   DATA[1132,29] := 12.07383;
   DATA[1132,30] := 1.724686;
   DATA[1132,31] := 1.274753;
   DATA[1132,32] := 0.7352687;
   DATA[1132,33] := 0.3084265;
   DATA[1132,34] := 2.0;
   DATA[1132,35] := 250.1442;
   DATA[1132,36] := 1.537821;
   DATA[1132,37] := 188.958;
   DATA[1132,38] := 0.000128152;
   DATA[1132,39] := 1.0;
   DATA[1133,0] := 2.551965;
   DATA[1133,1] := 721.1517;
   DATA[1133,2] := 2.0;
   DATA[1133,3] := 1.0;
   DATA[1133,4] := 262.5288;
   DATA[1133,5] := 8.463728;
   DATA[1133,6] := 316.7649;
   DATA[1133,8] := 1.0;
   DATA[1133,9] := 1.0;
   DATA[1133,10] := 1.0;
   DATA[1133,11] := 2.010372;
   DATA[1133,12] := 0.000256221;
   DATA[1133,13] := 1010.718;
   DATA[1133,14] := 1.0;
   DATA[1133,15] := 1.0;
   DATA[1133,16] := 1.0;
   DATA[1133,17] := 1.0;
   DATA[1133,18] := 1.0;
   DATA[1133,19] := 1.0;
   DATA[1133,20] := 148.808;
   DATA[1133,21] := 154.3963;
   DATA[1133,22] := 1.709672;
   DATA[1133,23] := 865.2397;
   DATA[1133,24] := 2.0;
   DATA[1133,25] := 2.0;
   DATA[1133,26] := 7.87798;
   DATA[1133,27] := 143.6042;
   DATA[1133,28] := 263.0095;
   DATA[1133,29] := 12.07383;
   DATA[1133,30] := 1.725455;
   DATA[1133,31] := 1.282567;
   DATA[1133,32] := 0.7352687;
   DATA[1133,33] := 0.3084265;
   DATA[1133,34] := 2.0;
   DATA[1133,35] := 250.1442;
   DATA[1133,36] := 1.69801;
   DATA[1133,37] := 189.1022;
   DATA[1133,38] := 0.000128152;
   DATA[1133,39] := 1.0;
   DATA[1134,0] := 2.548762;
   DATA[1134,1] := 722.604;
   DATA[1134,2] := 2.0;
   DATA[1134,3] := 1.0;
   DATA[1134,4] := 262.5288;
   DATA[1134,5] := 8.463728;
   DATA[1134,6] := 316.7649;
   DATA[1134,8] := 1.0;
   DATA[1134,9] := 1.0;
   DATA[1134,10] := 1.0;
   DATA[1134,11] := 2.010372;
   DATA[1134,12] := 0.000256221;
   DATA[1134,13] := 1010.959;
   DATA[1134,14] := 1.0;
   DATA[1134,15] := 1.0;
   DATA[1134,16] := 1.0;
   DATA[1134,17] := 1.0;
   DATA[1134,18] := 1.0;
   DATA[1134,19] := 1.0;
   DATA[1134,20] := 148.808;
   DATA[1134,21] := 154.3963;
   DATA[1134,22] := 1.709672;
   DATA[1134,23] := 865.1628;
   DATA[1134,24] := 2.0;
   DATA[1134,25] := 2.0;
   DATA[1134,26] := 7.87798;
   DATA[1134,27] := 143.6042;
   DATA[1134,28] := 263.0095;
   DATA[1134,29] := 12.07383;
   DATA[1134,30] := 1.725455;
   DATA[1134,31] := 1.282567;
   DATA[1134,32] := 0.7352687;
   DATA[1134,33] := 0.3084265;
   DATA[1134,34] := 2.0;
   DATA[1134,35] := 250.3044;
   DATA[1134,36] := 1.69801;
   DATA[1134,37] := 189.1662;
   DATA[1134,38] := 0.000128152;
   DATA[1134,39] := 1.0;
   DATA[1135,0] := 2.548762;
   DATA[1135,1] := 722.761;
   DATA[1135,2] := 2.0;
   DATA[1135,3] := 1.0;
   DATA[1135,4] := 262.5288;
   DATA[1135,5] := 8.463728;
   DATA[1135,6] := 316.7649;
   DATA[1135,8] := 1.0;
   DATA[1135,9] := 1.0;
   DATA[1135,10] := 1.0;
   DATA[1135,11] := 2.010372;
   DATA[1135,12] := 0.000256221;
   DATA[1135,13] := 1010.839;
   DATA[1135,14] := 1.0;
   DATA[1135,15] := 1.0;
   DATA[1135,16] := 1.0;
   DATA[1135,17] := 1.0;
   DATA[1135,18] := 1.0;
   DATA[1135,19] := 1.0;
   DATA[1135,20] := 148.808;
   DATA[1135,21] := 154.3963;
   DATA[1135,22] := 1.709672;
   DATA[1135,23] := 864.7398;
   DATA[1135,24] := 2.0;
   DATA[1135,25] := 2.0;
   DATA[1135,26] := 7.87798;
   DATA[1135,27] := 143.6042;
   DATA[1135,28] := 263.0095;
   DATA[1135,29] := 12.07383;
   DATA[1135,30] := 1.725455;
   DATA[1135,31] := 1.289484;
   DATA[1135,32] := 0.7352687;
   DATA[1135,33] := 0.3084265;
   DATA[1135,34] := 2.0;
   DATA[1135,35] := 250.3044;
   DATA[1135,36] := 1.69801;
   DATA[1135,37] := 189.1662;
   DATA[1135,38] := 0.000128152;
   DATA[1135,39] := 1.0;
   DATA[1136,0] := 2.548762;
   DATA[1136,1] := 723.4283;
   DATA[1136,2] := 2.0;
   DATA[1136,3] := 1.0;
   DATA[1136,4] := 262.5288;
   DATA[1136,5] := 8.463728;
   DATA[1136,6] := 316.97;
   DATA[1136,8] := 1.0;
   DATA[1136,9] := 1.0;
   DATA[1136,10] := 1.0;
   DATA[1136,11] := 2.010372;
   DATA[1136,12] := 0.000256221;
   DATA[1136,13] := 1011.039;
   DATA[1136,14] := 1.0;
   DATA[1136,15] := 1.0;
   DATA[1136,16] := 1.0;
   DATA[1136,17] := 1.0;
   DATA[1136,18] := 1.0;
   DATA[1136,19] := 1.0;
   DATA[1136,20] := 148.808;
   DATA[1136,21] := 154.3963;
   DATA[1136,22] := 1.709672;
   DATA[1136,23] := 864.586;
   DATA[1136,24] := 2.0;
   DATA[1136,25] := 2.0;
   DATA[1136,26] := 7.87798;
   DATA[1136,27] := 143.6042;
   DATA[1136,28] := 263.0095;
   DATA[1136,29] := 12.07383;
   DATA[1136,30] := 1.725455;
   DATA[1136,31] := 1.29243;
   DATA[1136,32] := 0.7352687;
   DATA[1136,33] := 0.3084265;
   DATA[1136,34] := 2.0;
   DATA[1136,35] := 250.3204;
   DATA[1136,36] := 1.69801;
   DATA[1136,37] := 189.1662;
   DATA[1136,38] := 0.000128152;
   DATA[1136,39] := 1.0;
   DATA[1137,0] := 2.548762;
   DATA[1137,1] := 723.8994;
   DATA[1137,2] := 2.0;
   DATA[1137,3] := 1.0;
   DATA[1137,4] := 262.5288;
   DATA[1137,5] := 8.463728;
   DATA[1137,6] := 316.97;
   DATA[1137,8] := 1.0;
   DATA[1137,9] := 1.0;
   DATA[1137,10] := 1.0;
   DATA[1137,11] := 2.010372;
   DATA[1137,12] := 0.000256221;
   DATA[1137,13] := 1010.959;
   DATA[1137,14] := 1.0;
   DATA[1137,15] := 1.0;
   DATA[1137,16] := 1.0;
   DATA[1137,17] := 1.0;
   DATA[1137,18] := 1.0;
   DATA[1137,19] := 1.0;
   DATA[1137,20] := 148.808;
   DATA[1137,21] := 154.3963;
   DATA[1137,22] := 1.712748;
   DATA[1137,23] := 864.0861;
   DATA[1137,24] := 2.0;
   DATA[1137,25] := 2.0;
   DATA[1137,26] := 7.87798;
   DATA[1137,27] := 143.6042;
   DATA[1137,28] := 263.0095;
   DATA[1137,29] := 12.07383;
   DATA[1137,30] := 1.725455;
   DATA[1137,31] := 1.29243;
   DATA[1137,32] := 0.7352687;
   DATA[1137,33] := 0.3084265;
   DATA[1137,34] := 2.0;
   DATA[1137,35] := 250.3204;
   DATA[1137,36] := 1.69801;
   DATA[1137,37] := 189.1662;
   DATA[1137,38] := 0.000128152;
   DATA[1137,39] := 1.0;
   DATA[1138,0] := 2.550364;
   DATA[1138,1] := 723.7424;
   DATA[1138,2] := 2.0;
   DATA[1138,3] := 1.0;
   DATA[1138,4] := 262.5288;
   DATA[1138,5] := 8.463728;
   DATA[1138,6] := 316.97;
   DATA[1138,8] := 1.0;
   DATA[1138,9] := 1.0;
   DATA[1138,10] := 1.0;
   DATA[1138,11] := 2.010372;
   DATA[1138,12] := 0.000256221;
   DATA[1138,13] := 1010.959;
   DATA[1138,14] := 1.0;
   DATA[1138,15] := 1.0;
   DATA[1138,16] := 1.0;
   DATA[1138,17] := 1.0;
   DATA[1138,18] := 1.0;
   DATA[1138,19] := 1.0;
   DATA[1138,20] := 148.808;
   DATA[1138,21] := 154.3963;
   DATA[1138,22] := 1.713389;
   DATA[1138,23] := 863.817;
   DATA[1138,24] := 2.0;
   DATA[1138,25] := 2.0;
   DATA[1138,26] := 7.87798;
   DATA[1138,27] := 143.6042;
   DATA[1138,28] := 263.0095;
   DATA[1138,29] := 12.07383;
   DATA[1138,30] := 1.725455;
   DATA[1138,31] := 1.285641;
   DATA[1138,32] := 0.7352687;
   DATA[1138,33] := 0.3084265;
   DATA[1138,34] := 2.0;
   DATA[1138,35] := 250.3204;
   DATA[1138,36] := 1.69801;
   DATA[1138,37] := 189.1662;
   DATA[1138,38] := 0.000128152;
   DATA[1138,39] := 1.0;
   DATA[1139,0] := 2.556449;
   DATA[1139,1] := 723.9386;
   DATA[1139,2] := 2.0;
   DATA[1139,3] := 1.0;
   DATA[1139,4] := 262.5288;
   DATA[1139,5] := 8.463728;
   DATA[1139,6] := 316.97;
   DATA[1139,8] := 1.0;
   DATA[1139,9] := 1.0;
   DATA[1139,10] := 1.0;
   DATA[1139,11] := 2.010372;
   DATA[1139,12] := 0.000256221;
   DATA[1139,13] := 1010.638;
   DATA[1139,14] := 1.0;
   DATA[1139,15] := 1.0;
   DATA[1139,16] := 1.0;
   DATA[1139,17] := 1.0;
   DATA[1139,18] := 1.0;
   DATA[1139,19] := 1.0;
   DATA[1139,20] := 148.808;
   DATA[1139,21] := 154.3963;
   DATA[1139,22] := 1.713389;
   DATA[1139,23] := 863.1248;
   DATA[1139,24] := 2.0;
   DATA[1139,25] := 2.0;
   DATA[1139,26] := 7.87798;
   DATA[1139,27] := 143.6042;
   DATA[1139,28] := 263.0095;
   DATA[1139,29] := 12.07383;
   DATA[1139,30] := 1.725455;
   DATA[1139,31] := 1.282311;
   DATA[1139,32] := 0.7352687;
   DATA[1139,33] := 0.3084265;
   DATA[1139,34] := 2.0;
   DATA[1139,35] := 250.2724;
   DATA[1139,36] := 1.69801;
   DATA[1139,37] := 189.0541;
   DATA[1139,38] := 0.000128152;
   DATA[1139,39] := 1.0;
   DATA[1140,0] := 2.560292;
   DATA[1140,1] := 724.9199;
   DATA[1140,2] := 2.0;
   DATA[1140,3] := 1.0;
   DATA[1140,4] := 262.5288;
   DATA[1140,5] := 8.463728;
   DATA[1140,6] := 316.97;
   DATA[1140,8] := 1.0;
   DATA[1140,9] := 1.0;
   DATA[1140,10] := 1.0;
   DATA[1140,11] := 2.010372;
   DATA[1140,12] := 0.000256221;
   DATA[1140,13] := 1011.039;
   DATA[1140,14] := 1.0;
   DATA[1140,15] := 1.0;
   DATA[1140,16] := 1.0;
   DATA[1140,17] := 1.0;
   DATA[1140,18] := 1.0;
   DATA[1140,19] := 1.0;
   DATA[1140,20] := 148.808;
   DATA[1140,21] := 154.3963;
   DATA[1140,22] := 1.713389;
   DATA[1140,23] := 862.8172;
   DATA[1140,24] := 2.0;
   DATA[1140,25] := 2.0;
   DATA[1140,26] := 7.87798;
   DATA[1140,27] := 143.6042;
   DATA[1140,28] := 263.0095;
   DATA[1140,29] := 12.07383;
   DATA[1140,30] := 1.725455;
   DATA[1140,31] := 1.264891;
   DATA[1140,32] := 0.7352687;
   DATA[1140,33] := 0.3084265;
   DATA[1140,34] := 2.0;
   DATA[1140,35] := 250.1762;
   DATA[1140,36] := 1.69801;
   DATA[1140,37] := 189.0541;
   DATA[1140,38] := 0.000128152;
   DATA[1140,39] := 1.0;
   DATA[1141,0] := 2.560292;
   DATA[1141,1] := 725.1555;
   DATA[1141,2] := 2.0;
   DATA[1141,3] := 1.0;
   DATA[1141,4] := 262.5288;
   DATA[1141,5] := 8.463728;
   DATA[1141,6] := 316.97;
   DATA[1141,8] := 1.0;
   DATA[1141,9] := 1.0;
   DATA[1141,10] := 1.0;
   DATA[1141,11] := 2.010372;
   DATA[1141,12] := 0.000256221;
   DATA[1141,13] := 1010.678;
   DATA[1141,14] := 1.0;
   DATA[1141,15] := 1.0;
   DATA[1141,16] := 1.0;
   DATA[1141,17] := 1.0;
   DATA[1141,18] := 1.0;
   DATA[1141,19] := 1.0;
   DATA[1141,20] := 148.808;
   DATA[1141,21] := 154.3963;
   DATA[1141,22] := 1.713389;
   DATA[1141,23] := 862.548;
   DATA[1141,24] := 2.0;
   DATA[1141,25] := 2.0;
   DATA[1141,26] := 7.87798;
   DATA[1141,27] := 143.6042;
   DATA[1141,28] := 263.0095;
   DATA[1141,29] := 12.07383;
   DATA[1141,30] := 1.725455;
   DATA[1141,31] := 1.264634;
   DATA[1141,32] := 0.7352687;
   DATA[1141,33] := 0.3084265;
   DATA[1141,34] := 2.0;
   DATA[1141,35] := 250.1762;
   DATA[1141,36] := 1.69801;
   DATA[1141,37] := 189.0541;
   DATA[1141,38] := 0.000128152;
   DATA[1141,39] := 1.0;
   DATA[1142,0] := 2.560292;
   DATA[1142,1] := 725.7835;
   DATA[1142,2] := 2.0;
   DATA[1142,3] := 1.0;
   DATA[1142,4] := 262.5288;
   DATA[1142,5] := 8.463728;
   DATA[1142,6] := 316.97;
   DATA[1142,8] := 1.0;
   DATA[1142,9] := 1.0;
   DATA[1142,10] := 1.0;
   DATA[1142,11] := 2.010372;
   DATA[1142,12] := 0.000256221;
   DATA[1142,13] := 1011.119;
   DATA[1142,14] := 1.0;
   DATA[1142,15] := 1.0;
   DATA[1142,16] := 1.0;
   DATA[1142,17] := 1.0;
   DATA[1142,18] := 1.0;
   DATA[1142,19] := 1.0;
   DATA[1142,20] := 148.808;
   DATA[1142,21] := 154.3963;
   DATA[1142,22] := 1.714029;
   DATA[1142,23] := 862.0867;
   DATA[1142,24] := 2.0;
   DATA[1142,25] := 2.0;
   DATA[1142,26] := 7.87798;
   DATA[1142,27] := 143.6042;
   DATA[1142,28] := 263.0095;
   DATA[1142,29] := 12.07383;
   DATA[1142,30] := 1.725455;
   DATA[1142,31] := 1.272064;
   DATA[1142,32] := 0.7352687;
   DATA[1142,33] := 0.3084265;
   DATA[1142,34] := 2.0;
   DATA[1142,35] := 250.3204;
   DATA[1142,36] := 1.69801;
   DATA[1142,37] := 189.0541;
   DATA[1142,38] := 0.000128152;
   DATA[1142,39] := 1.0;
   DATA[1143,0] := 2.560292;
   DATA[1143,1] := 726.4901;
   DATA[1143,2] := 2.0;
   DATA[1143,3] := 1.0;
   DATA[1143,4] := 262.5288;
   DATA[1143,5] := 8.463728;
   DATA[1143,6] := 316.9187;
   DATA[1143,8] := 1.0;
   DATA[1143,9] := 1.0;
   DATA[1143,10] := 1.0;
   DATA[1143,11] := 2.010372;
   DATA[1143,12] := 0.000256221;
   DATA[1143,13] := 1011.159;
   DATA[1143,14] := 1.0;
   DATA[1143,15] := 1.0;
   DATA[1143,16] := 1.0;
   DATA[1143,17] := 1.0;
   DATA[1143,18] := 1.0;
   DATA[1143,19] := 1.0;
   DATA[1143,20] := 148.808;
   DATA[1143,21] := 154.3963;
   DATA[1143,22] := 1.714798;
   DATA[1143,23] := 862.0867;
   DATA[1143,24] := 2.0;
   DATA[1143,25] := 2.0;
   DATA[1143,26] := 7.87798;
   DATA[1143,27] := 143.6042;
   DATA[1143,28] := 263.0095;
   DATA[1143,29] := 12.07383;
   DATA[1143,30] := 1.725455;
   DATA[1143,31] := 1.272064;
   DATA[1143,32] := 0.7357808;
   DATA[1143,33] := 0.3084265;
   DATA[1143,34] := 2.0;
   DATA[1143,35] := 250.3365;
   DATA[1143,36] := 1.69801;
   DATA[1143,37] := 189.1823;
   DATA[1143,38] := 0.000128152;
   DATA[1143,39] := 1.0;
   DATA[1144,0] := 2.551324;
   DATA[1144,1] := 726.9218;
   DATA[1144,2] := 2.0;
   DATA[1144,3] := 1.0;
   DATA[1144,4] := 262.5288;
   DATA[1144,5] := 8.463728;
   DATA[1144,6] := 316.7649;
   DATA[1144,8] := 1.0;
   DATA[1144,9] := 1.0;
   DATA[1144,10] := 1.0;
   DATA[1144,11] := 2.010372;
   DATA[1144,12] := 0.000256221;
   DATA[1144,13] := 1011.279;
   DATA[1144,14] := 1.0;
   DATA[1144,15] := 1.0;
   DATA[1144,16] := 1.0;
   DATA[1144,17] := 1.0;
   DATA[1144,18] := 1.0;
   DATA[1144,19] := 1.0;
   DATA[1144,20] := 148.808;
   DATA[1144,21] := 154.3963;
   DATA[1144,22] := 1.714029;
   DATA[1144,23] := 861.6252;
   DATA[1144,24] := 2.0;
   DATA[1144,25] := 2.0;
   DATA[1144,26] := 7.87798;
   DATA[1144,27] := 143.6042;
   DATA[1144,28] := 263.0095;
   DATA[1144,29] := 12.07383;
   DATA[1144,30] := 1.725455;
   DATA[1144,31] := 1.288075;
   DATA[1144,32] := 0.7379573;
   DATA[1144,33] := 0.3084265;
   DATA[1144,34] := 2.0;
   DATA[1144,35] := 250.3365;
   DATA[1144,36] := 1.69801;
   DATA[1144,37] := 189.3265;
   DATA[1144,38] := 0.000128152;
   DATA[1144,39] := 1.0;
   DATA[1145,0] := 2.544919;
   DATA[1145,1] := 727.3143;
   DATA[1145,2] := 2.0;
   DATA[1145,3] := 1.0;
   DATA[1145,4] := 262.5288;
   DATA[1145,5] := 8.463728;
   DATA[1145,6] := 316.7649;
   DATA[1145,8] := 1.0;
   DATA[1145,9] := 1.0;
   DATA[1145,10] := 1.0;
   DATA[1145,11] := 2.010372;
   DATA[1145,12] := 0.000256221;
   DATA[1145,13] := 1011.279;
   DATA[1145,14] := 1.0;
   DATA[1145,15] := 1.0;
   DATA[1145,16] := 1.0;
   DATA[1145,17] := 1.0;
   DATA[1145,18] := 1.0;
   DATA[1145,19] := 1.0;
   DATA[1145,20] := 148.808;
   DATA[1145,21] := 154.3963;
   DATA[1145,22] := 1.713261;
   DATA[1145,23] := 861.3945;
   DATA[1145,24] := 2.0;
   DATA[1145,25] := 2.0;
   DATA[1145,26] := 7.87798;
   DATA[1145,27] := 143.6042;
   DATA[1145,28] := 263.0095;
   DATA[1145,29] := 12.07383;
   DATA[1145,30] := 1.725711;
   DATA[1145,31] := 1.28641;
   DATA[1145,32] := 0.7379573;
   DATA[1145,33] := 0.3084265;
   DATA[1145,34] := 2.0;
   DATA[1145,35] := 250.3365;
   DATA[1145,36] := 1.69801;
   DATA[1145,37] := 189.3265;
   DATA[1145,38] := 0.000128152;
   DATA[1145,39] := 1.0;
   DATA[1146,0] := 2.539154;
   DATA[1146,1] := 727.9424;
   DATA[1146,2] := 2.0;
   DATA[1146,3] := 1.0;
   DATA[1146,4] := 262.5288;
   DATA[1146,5] := 8.463728;
   DATA[1146,6] := 316.7649;
   DATA[1146,8] := 1.0;
   DATA[1146,9] := 1.0;
   DATA[1146,10] := 1.0;
   DATA[1146,11] := 2.010372;
   DATA[1146,12] := 0.000256221;
   DATA[1146,13] := 1011.439;
   DATA[1146,14] := 1.0;
   DATA[1146,15] := 1.0;
   DATA[1146,16] := 1.0;
   DATA[1146,17] := 1.0;
   DATA[1146,18] := 1.0;
   DATA[1146,19] := 1.0;
   DATA[1146,20] := 148.808;
   DATA[1146,21] := 154.3963;
   DATA[1146,22] := 1.713261;
   DATA[1146,23] := 861.2407;
   DATA[1146,24] := 2.0;
   DATA[1146,25] := 2.0;
   DATA[1146,26] := 7.87798;
   DATA[1146,27] := 143.6042;
   DATA[1146,28] := 263.0095;
   DATA[1146,29] := 12.07383;
   DATA[1146,30] := 1.726609;
   DATA[1146,31] := 1.286794;
   DATA[1146,32] := 0.7379573;
   DATA[1146,33] := 0.3084265;
   DATA[1146,34] := 2.0;
   DATA[1146,35] := 250.3365;
   DATA[1146,36] := 1.69801;
   DATA[1146,37] := 189.3265;
   DATA[1146,38] := 0.000128152;
   DATA[1146,39] := 1.0;
   DATA[1147,0] := 2.539154;
   DATA[1147,1] := 728.0602;
   DATA[1147,2] := 2.0;
   DATA[1147,3] := 1.0;
   DATA[1147,4] := 262.5288;
   DATA[1147,5] := 8.463728;
   DATA[1147,6] := 316.7649;
   DATA[1147,8] := 1.0;
   DATA[1147,9] := 1.0;
   DATA[1147,10] := 1.0;
   DATA[1147,11] := 2.010372;
   DATA[1147,12] := 0.000256221;
   DATA[1147,13] := 1011.239;
   DATA[1147,14] := 1.0;
   DATA[1147,15] := 1.0;
   DATA[1147,16] := 1.0;
   DATA[1147,17] := 1.0;
   DATA[1147,18] := 1.0;
   DATA[1147,19] := 1.0;
   DATA[1147,20] := 148.808;
   DATA[1147,21] := 154.3963;
   DATA[1147,22] := 1.714926;
   DATA[1147,23] := 860.4332;
   DATA[1147,24] := 2.0;
   DATA[1147,25] := 2.0;
   DATA[1147,26] := 7.87798;
   DATA[1147,27] := 143.6042;
   DATA[1147,28] := 263.0095;
   DATA[1147,29] := 12.07383;
   DATA[1147,30] := 1.726609;
   DATA[1147,31] := 1.292558;
   DATA[1147,32] := 0.7348846;
   DATA[1147,33] := 0.3084265;
   DATA[1147,34] := 2.0;
   DATA[1147,35] := 250.3365;
   DATA[1147,36] := 1.69801;
   DATA[1147,37] := 189.1342;
   DATA[1147,38] := 0.000128152;
   DATA[1147,39] := 1.0;
   DATA[1148,0] := 2.539154;
   DATA[1148,1] := 728.6882;
   DATA[1148,2] := 2.0;
   DATA[1148,3] := 1.0;
   DATA[1148,4] := 262.5288;
   DATA[1148,5] := 8.463728;
   DATA[1148,6] := 316.97;
   DATA[1148,8] := 1.0;
   DATA[1148,9] := 1.0;
   DATA[1148,10] := 1.0;
   DATA[1148,11] := 2.010372;
   DATA[1148,12] := 0.000256221;
   DATA[1148,13] := 1011.159;
   DATA[1148,14] := 1.0;
   DATA[1148,15] := 1.0;
   DATA[1148,16] := 1.0;
   DATA[1148,17] := 1.0;
   DATA[1148,18] := 1.0;
   DATA[1148,19] := 1.0;
   DATA[1148,20] := 148.808;
   DATA[1148,21] := 154.3963;
   DATA[1148,22] := 1.715952;
   DATA[1148,23] := 859.7795;
   DATA[1148,24] := 2.0;
   DATA[1148,25] := 2.0;
   DATA[1148,26] := 7.87798;
   DATA[1148,27] := 143.6042;
   DATA[1148,28] := 263.0095;
   DATA[1148,29] := 12.07383;
   DATA[1148,30] := 1.726609;
   DATA[1148,31] := 1.292558;
   DATA[1148,32] := 0.7348846;
   DATA[1148,33] := 0.3084265;
   DATA[1148,34] := 2.0;
   DATA[1148,35] := 250.3365;
   DATA[1148,36] := 1.69801;
   DATA[1148,37] := 189.1182;
   DATA[1148,38] := 0.000128152;
   DATA[1148,39] := 1.0;
   DATA[1149,0] := 2.539154;
   DATA[1149,1] := 729.2377;
   DATA[1149,2] := 2.0;
   DATA[1149,3] := 1.0;
   DATA[1149,4] := 262.5288;
   DATA[1149,5] := 8.467573;
   DATA[1149,6] := 316.97;
   DATA[1149,8] := 1.0;
   DATA[1149,9] := 1.0;
   DATA[1149,10] := 1.0;
   DATA[1149,11] := 2.010372;
   DATA[1149,12] := 0.000256221;
   DATA[1149,13] := 1011.119;
   DATA[1149,14] := 1.0;
   DATA[1149,15] := 1.0;
   DATA[1149,16] := 1.0;
   DATA[1149,17] := 1.0;
   DATA[1149,18] := 1.0;
   DATA[1149,19] := 1.0;
   DATA[1149,20] := 148.808;
   DATA[1149,21] := 154.3963;
   DATA[1149,22] := 1.715952;
   DATA[1149,23] := 859.5873;
   DATA[1149,24] := 2.0;
   DATA[1149,25] := 2.0;
   DATA[1149,26] := 7.87798;
   DATA[1149,27] := 143.6042;
   DATA[1149,28] := 263.0095;
   DATA[1149,29] := 12.07383;
   DATA[1149,30] := 1.726609;
   DATA[1149,31] := 1.301012;
   DATA[1149,32] := 0.7348846;
   DATA[1149,33] := 0.3084265;
   DATA[1149,34] := 2.0;
   DATA[1149,35] := 250.3365;
   DATA[1149,36] := 1.69801;
   DATA[1149,37] := 189.1182;
   DATA[1149,38] := 0.000128152;
   DATA[1149,39] := 1.0;
   DATA[1150,0] := 2.54684;
   DATA[1150,1] := 729.8658;
   DATA[1150,2] := 2.0;
   DATA[1150,3] := 1.0;
   DATA[1150,4] := 262.5288;
   DATA[1150,5] := 8.467573;
   DATA[1150,6] := 316.97;
   DATA[1150,8] := 1.0;
   DATA[1150,9] := 1.0;
   DATA[1150,10] := 1.0;
   DATA[1150,11] := 2.010372;
   DATA[1150,12] := 0.000256221;
   DATA[1150,13] := 1011.079;
   DATA[1150,14] := 1.0;
   DATA[1150,15] := 1.0;
   DATA[1150,16] := 1.0;
   DATA[1150,17] := 1.0;
   DATA[1150,18] := 1.0;
   DATA[1150,19] := 1.0;
   DATA[1150,20] := 148.808;
   DATA[1150,21] := 154.3963;
   DATA[1150,22] := 1.715952;
   DATA[1150,23] := 858.972;
   DATA[1150,24] := 2.0;
   DATA[1150,25] := 2.0;
   DATA[1150,26] := 7.87798;
   DATA[1150,27] := 143.6042;
   DATA[1150,28] := 263.0095;
   DATA[1150,29] := 12.07383;
   DATA[1150,30] := 1.726609;
   DATA[1150,31] := 1.294607;
   DATA[1150,32] := 0.7348846;
   DATA[1150,33] := 0.3084265;
   DATA[1150,34] := 2.0;
   DATA[1150,35] := 250.3365;
   DATA[1150,36] := 1.69801;
   DATA[1150,37] := 189.1182;
   DATA[1150,38] := 0.000128152;
   DATA[1150,39] := 1.0;
   DATA[1151,0] := 2.547481;
   DATA[1151,1] := 729.905;
   DATA[1151,2] := 2.0;
   DATA[1151,3] := 1.0;
   DATA[1151,4] := 262.5288;
   DATA[1151,5] := 8.467573;
   DATA[1151,6] := 316.97;
   DATA[1151,8] := 1.0;
   DATA[1151,9] := 1.0;
   DATA[1151,10] := 1.0;
   DATA[1151,11] := 2.010372;
   DATA[1151,12] := 0.000256221;
   DATA[1151,13] := 1011.079;
   DATA[1151,14] := 1.0;
   DATA[1151,15] := 1.0;
   DATA[1151,16] := 1.0;
   DATA[1151,17] := 1.0;
   DATA[1151,18] := 1.0;
   DATA[1151,19] := 1.0;
   DATA[1151,20] := 148.808;
   DATA[1151,21] := 154.3963;
   DATA[1151,22] := 1.715952;
   DATA[1151,23] := 858.7029;
   DATA[1151,24] := 2.0;
   DATA[1151,25] := 2.0;
   DATA[1151,26] := 7.87798;
   DATA[1151,27] := 143.6042;
   DATA[1151,28] := 263.0095;
   DATA[1151,29] := 12.07383;
   DATA[1151,30] := 1.726609;
   DATA[1151,31] := 1.288971;
   DATA[1151,32] := 0.7348846;
   DATA[1151,33] := 0.3084265;
   DATA[1151,34] := 2.0;
   DATA[1151,35] := 250.3365;
   DATA[1151,36] := 1.69801;
   DATA[1151,37] := 189.2944;
   DATA[1151,38] := 0.000128152;
   DATA[1151,39] := 1.0;
   DATA[1152,0] := 2.552926;
   DATA[1152,1] := 730.1013;
   DATA[1152,2] := 2.0;
   DATA[1152,3] := 1.0;
   DATA[1152,4] := 262.5288;
   DATA[1152,5] := 8.467573;
   DATA[1152,6] := 316.97;
   DATA[1152,8] := 1.0;
   DATA[1152,9] := 1.0;
   DATA[1152,10] := 1.0;
   DATA[1152,11] := 2.010372;
   DATA[1152,12] := 0.000256221;
   DATA[1152,13] := 1010.959;
   DATA[1152,14] := 1.0;
   DATA[1152,15] := 1.0;
   DATA[1152,16] := 1.0;
   DATA[1152,17] := 1.0;
   DATA[1152,18] := 1.0;
   DATA[1152,19] := 1.0;
   DATA[1152,20] := 148.808;
   DATA[1152,21] := 154.3963;
   DATA[1152,22] := 1.71608;
   DATA[1152,23] := 858.3184;
   DATA[1152,24] := 2.0;
   DATA[1152,25] := 2.0;
   DATA[1152,26] := 7.87798;
   DATA[1152,27] := 143.6042;
   DATA[1152,28] := 263.0095;
   DATA[1152,29] := 12.07383;
   DATA[1152,30] := 1.726609;
   DATA[1152,31] := 1.276803;
   DATA[1152,32] := 0.7348846;
   DATA[1152,33] := 0.3084265;
   DATA[1152,34] := 2.0;
   DATA[1152,35] := 250.5127;
   DATA[1152,36] := 1.69801;
   DATA[1152,37] := 189.2944;
   DATA[1152,38] := 0.000128152;
   DATA[1152,39] := 1.0;
   DATA[1153,0] := 2.553566;
   DATA[1153,1] := 731.2396;
   DATA[1153,2] := 2.0;
   DATA[1153,3] := 1.0;
   DATA[1153,4] := 262.5288;
   DATA[1153,5] := 8.467573;
   DATA[1153,6] := 316.97;
   DATA[1153,8] := 1.0;
   DATA[1153,9] := 1.0;
   DATA[1153,10] := 1.0;
   DATA[1153,11] := 2.010372;
   DATA[1153,12] := 0.000256221;
   DATA[1153,13] := 1011.159;
   DATA[1153,14] := 1.0;
   DATA[1153,15] := 1.0;
   DATA[1153,16] := 1.0;
   DATA[1153,17] := 1.0;
   DATA[1153,18] := 1.0;
   DATA[1153,19] := 1.0;
   DATA[1153,20] := 148.808;
   DATA[1153,21] := 154.3963;
   DATA[1153,22] := 1.717746;
   DATA[1153,23] := 857.5493;
   DATA[1153,24] := 2.0;
   DATA[1153,25] := 2.0;
   DATA[1153,26] := 7.87798;
   DATA[1153,27] := 143.6042;
   DATA[1153,28] := 263.0095;
   DATA[1153,29] := 12.07383;
   DATA[1153,30] := 1.726609;
   DATA[1153,31] := 1.27296;
   DATA[1153,32] := 0.7348846;
   DATA[1153,33] := 0.3084265;
   DATA[1153,34] := 2.0;
   DATA[1153,35] := 250.5127;
   DATA[1153,36] := 1.69801;
   DATA[1153,37] := 189.2944;
   DATA[1153,38] := 0.000128152;
   DATA[1153,39] := 1.0;
   DATA[1154,0] := 2.553566;
   DATA[1154,1] := 731.2396;
   DATA[1154,2] := 2.0;
   DATA[1154,3] := 1.0;
   DATA[1154,4] := 262.5288;
   DATA[1154,5] := 8.467573;
   DATA[1154,6] := 316.97;
   DATA[1154,8] := 1.0;
   DATA[1154,9] := 1.0;
   DATA[1154,10] := 1.0;
   DATA[1154,11] := 2.010372;
   DATA[1154,12] := 0.000256221;
   DATA[1154,13] := 1011.159;
   DATA[1154,14] := 1.0;
   DATA[1154,15] := 1.0;
   DATA[1154,16] := 1.0;
   DATA[1154,17] := 1.0;
   DATA[1154,18] := 1.0;
   DATA[1154,19] := 1.0;
   DATA[1154,20] := 148.808;
   DATA[1154,21] := 154.3963;
   DATA[1154,22] := 1.717746;
   DATA[1154,23] := 857.5493;
   DATA[1154,24] := 2.0;
   DATA[1154,25] := 2.0;
   DATA[1154,26] := 7.87798;
   DATA[1154,27] := 143.6042;
   DATA[1154,28] := 263.0095;
   DATA[1154,29] := 12.07383;
   DATA[1154,30] := 1.726609;
   DATA[1154,31] := 1.27296;
   DATA[1154,32] := 0.7348846;
   DATA[1154,33] := 0.3084265;
   DATA[1154,34] := 2.0;
   DATA[1154,35] := 250.5127;
   DATA[1154,36] := 1.69801;
   DATA[1154,37] := 189.2944;
   DATA[1154,38] := 0.000128152;
   DATA[1154,39] := 1.0;
   DATA[1155,0] := 2.556129;
   DATA[1155,1] := 731.3967;
   DATA[1155,2] := 2.0;
   DATA[1155,3] := 1.0;
   DATA[1155,4] := 262.5288;
   DATA[1155,5] := 8.467573;
   DATA[1155,6] := 316.97;
   DATA[1155,8] := 1.0;
   DATA[1155,9] := 1.0;
   DATA[1155,10] := 1.0;
   DATA[1155,11] := 2.010372;
   DATA[1155,12] := 0.000256221;
   DATA[1155,13] := 1011.279;
   DATA[1155,14] := 1.0;
   DATA[1155,15] := 1.0;
   DATA[1155,16] := 1.0;
   DATA[1155,17] := 1.0;
   DATA[1155,18] := 1.0;
   DATA[1155,19] := 1.0;
   DATA[1155,20] := 148.808;
   DATA[1155,21] := 154.3963;
   DATA[1155,22] := 1.718515;
   DATA[1155,23] := 857.5493;
   DATA[1155,24] := 2.0;
   DATA[1155,25] := 2.0;
   DATA[1155,26] := 7.87798;
   DATA[1155,27] := 143.6042;
   DATA[1155,28] := 263.0095;
   DATA[1155,29] := 12.07383;
   DATA[1155,30] := 1.726609;
   DATA[1155,31] := 1.281158;
   DATA[1155,32] := 0.7348846;
   DATA[1155,33] := 0.3072094;
   DATA[1155,34] := 2.0;
   DATA[1155,35] := 250.5447;
   DATA[1155,36] := 1.69801;
   DATA[1155,37] := 189.2944;
   DATA[1155,38] := 0.000128152;
   DATA[1155,39] := 1.0;
   DATA[1156,0] := 2.556129;
   DATA[1156,1] := 731.9462;
   DATA[1156,2] := 2.0;
   DATA[1156,3] := 1.0;
   DATA[1156,4] := 262.5288;
   DATA[1156,5] := 8.467573;
   DATA[1156,6] := 316.97;
   DATA[1156,8] := 1.0;
   DATA[1156,9] := 1.0;
   DATA[1156,10] := 1.0;
   DATA[1156,11] := 2.010372;
   DATA[1156,12] := 0.000256221;
   DATA[1156,13] := 1011.359;
   DATA[1156,14] := 1.0;
   DATA[1156,15] := 1.0;
   DATA[1156,16] := 1.0;
   DATA[1156,17] := 1.0;
   DATA[1156,18] := 1.0;
   DATA[1156,19] := 1.0;
   DATA[1156,20] := 148.808;
   DATA[1156,21] := 154.3963;
   DATA[1156,22] := 1.718515;
   DATA[1156,23] := 857.2033;
   DATA[1156,24] := 2.0;
   DATA[1156,25] := 2.0;
   DATA[1156,26] := 7.87798;
   DATA[1156,27] := 143.6042;
   DATA[1156,28] := 263.0095;
   DATA[1156,29] := 12.07383;
   DATA[1156,30] := 1.726609;
   DATA[1156,31] := 1.282823;
   DATA[1156,32] := 0.7361649;
   DATA[1156,33] := 0.3084905;
   DATA[1156,34] := 2.0;
   DATA[1156,35] := 250.5447;
   DATA[1156,36] := 1.69801;
   DATA[1156,37] := 189.2944;
   DATA[1156,38] := 0.000128152;
   DATA[1156,39] := 1.0;
   DATA[1157,0] := 2.556129;
   DATA[1157,1] := 732.535;
   DATA[1157,2] := 2.0;
   DATA[1157,3] := 1.0;
   DATA[1157,4] := 262.5288;
   DATA[1157,5] := 8.467573;
   DATA[1157,6] := 316.97;
   DATA[1157,8] := 1.0;
   DATA[1157,9] := 1.0;
   DATA[1157,10] := 1.0;
   DATA[1157,11] := 2.010372;
   DATA[1157,12] := 0.000256221;
   DATA[1157,13] := 1010.959;
   DATA[1157,14] := 1.0;
   DATA[1157,15] := 1.0;
   DATA[1157,16] := 1.0;
   DATA[1157,17] := 1.0;
   DATA[1157,18] := 1.0;
   DATA[1157,19] := 1.0;
   DATA[1157,20] := 148.808;
   DATA[1157,21] := 154.3963;
   DATA[1157,22] := 1.719027;
   DATA[1157,23] := 856.7803;
   DATA[1157,24] := 2.0;
   DATA[1157,25] := 2.0;
   DATA[1157,26] := 7.87798;
   DATA[1157,27] := 143.6042;
   DATA[1157,28] := 263.0095;
   DATA[1157,29] := 12.07383;
   DATA[1157,30] := 1.726609;
   DATA[1157,31] := 1.291789;
   DATA[1157,32] := 0.7361649;
   DATA[1157,33] := 0.3084905;
   DATA[1157,34] := 2.0;
   DATA[1157,35] := 250.5447;
   DATA[1157,36] := 1.69801;
   DATA[1157,37] := 189.2944;
   DATA[1157,38] := 0.000128152;
   DATA[1157,39] := 1.0;
   DATA[1158,0] := 2.556129;
   DATA[1158,1] := 732.8098;
   DATA[1158,2] := 2.0;
   DATA[1158,3] := 1.0;
   DATA[1158,4] := 262.5288;
   DATA[1158,5] := 8.467573;
   DATA[1158,6] := 316.97;
   DATA[1158,8] := 1.0;
   DATA[1158,9] := 1.0;
   DATA[1158,10] := 1.0;
   DATA[1158,11] := 2.010372;
   DATA[1158,12] := 0.000256221;
   DATA[1158,13] := 1011.479;
   DATA[1158,14] := 1.0;
   DATA[1158,15] := 1.0;
   DATA[1158,16] := 1.0;
   DATA[1158,17] := 1.0;
   DATA[1158,18] := 1.0;
   DATA[1158,19] := 1.0;
   DATA[1158,20] := 148.808;
   DATA[1158,21] := 154.3963;
   DATA[1158,22] := 1.719027;
   DATA[1158,23] := 856.0882;
   DATA[1158,24] := 2.0;
   DATA[1158,25] := 2.0;
   DATA[1158,26] := 7.87798;
   DATA[1158,27] := 143.6042;
   DATA[1158,28] := 263.0095;
   DATA[1158,29] := 12.07383;
   DATA[1158,30] := 1.726609;
   DATA[1158,31] := 1.291789;
   DATA[1158,32] := 0.7357808;
   DATA[1158,33] := 0.3084905;
   DATA[1158,34] := 2.0;
   DATA[1158,35] := 250.5447;
   DATA[1158,36] := 1.649953;
   DATA[1158,37] := 189.2944;
   DATA[1158,38] := 0.000128152;
   DATA[1158,39] := 1.0;
   DATA[1159,0] := 2.547161;
   DATA[1159,1] := 733.32;
   DATA[1159,2] := 2.0;
   DATA[1159,3] := 1.0;
   DATA[1159,4] := 262.5288;
   DATA[1159,5] := 8.467573;
   DATA[1159,6] := 316.97;
   DATA[1159,8] := 1.0;
   DATA[1159,9] := 1.0;
   DATA[1159,10] := 1.0;
   DATA[1159,11] := 2.010372;
   DATA[1159,12] := 0.000256221;
   DATA[1159,13] := 1011.039;
   DATA[1159,14] := 1.0;
   DATA[1159,15] := 1.0;
   DATA[1159,16] := 1.0;
   DATA[1159,17] := 1.0;
   DATA[1159,18] := 1.0;
   DATA[1159,19] := 1.0;
   DATA[1159,20] := 148.808;
   DATA[1159,21] := 154.3963;
   DATA[1159,22] := 1.717105;
   DATA[1159,23] := 855.3576;
   DATA[1159,24] := 2.0;
   DATA[1159,25] := 2.0;
   DATA[1159,26] := 7.87798;
   DATA[1159,27] := 143.6042;
   DATA[1159,28] := 263.0095;
   DATA[1159,29] := 12.07383;
   DATA[1159,30] := 1.724942;
   DATA[1159,31] := 1.291789;
   DATA[1159,32] := 0.7347566;
   DATA[1159,33] := 0.3084905;
   DATA[1159,34] := 2.0;
   DATA[1159,35] := 250.5447;
   DATA[1159,36] := 1.649953;
   DATA[1159,37] := 189.2944;
   DATA[1159,38] := 0.000128152;
   DATA[1159,39] := 1.0;
   DATA[1160,0] := 2.545239;
   DATA[1160,1] := 733.634;
   DATA[1160,2] := 2.0;
   DATA[1160,3] := 1.0;
   DATA[1160,4] := 262.5288;
   DATA[1160,5] := 8.467573;
   DATA[1160,6] := 316.97;
   DATA[1160,8] := 1.0;
   DATA[1160,9] := 1.0;
   DATA[1160,10] := 1.0;
   DATA[1160,11] := 2.010372;
   DATA[1160,12] := 0.000256221;
   DATA[1160,13] := 1011.039;
   DATA[1160,14] := 1.0;
   DATA[1160,15] := 1.0;
   DATA[1160,16] := 1.0;
   DATA[1160,17] := 1.0;
   DATA[1160,18] := 1.0;
   DATA[1160,19] := 1.0;
   DATA[1160,20] := 148.808;
   DATA[1160,21] := 154.3963;
   DATA[1160,22] := 1.715824;
   DATA[1160,23] := 855.2422;
   DATA[1160,24] := 2.0;
   DATA[1160,25] := 2.0;
   DATA[1160,26] := 7.87798;
   DATA[1160,27] := 143.6042;
   DATA[1160,28] := 263.0095;
   DATA[1160,29] := 12.07383;
   DATA[1160,30] := 1.724942;
   DATA[1160,31] := 1.308057;
   DATA[1160,32] := 0.7347566;
   DATA[1160,33] := 0.3084905;
   DATA[1160,34] := 2.0;
   DATA[1160,35] := 250.4326;
   DATA[1160,36] := 1.649953;
   DATA[1160,37] := 189.2944;
   DATA[1160,38] := 0.000128152;
   DATA[1160,39] := 1.0;
   DATA[1161,0] := 2.543638;
   DATA[1161,1] := 733.4378;
   DATA[1161,2] := 2.0;
   DATA[1161,3] := 1.0;
   DATA[1161,4] := 262.5288;
   DATA[1161,5] := 8.467573;
   DATA[1161,6] := 316.97;
   DATA[1161,8] := 1.0;
   DATA[1161,9] := 1.0;
   DATA[1161,10] := 1.0;
   DATA[1161,11] := 2.010372;
   DATA[1161,12] := 0.000256221;
   DATA[1161,13] := 1010.839;
   DATA[1161,14] := 1.0;
   DATA[1161,15] := 1.0;
   DATA[1161,16] := 1.0;
   DATA[1161,17] := 1.0;
   DATA[1161,18] := 1.0;
   DATA[1161,19] := 1.0;
   DATA[1161,20] := 148.808;
   DATA[1161,21] := 154.3963;
   DATA[1161,22] := 1.715824;
   DATA[1161,23] := 855.05;
   DATA[1161,24] := 2.0;
   DATA[1161,25] := 2.0;
   DATA[1161,26] := 7.87798;
   DATA[1161,27] := 143.6042;
   DATA[1161,28] := 263.0095;
   DATA[1161,29] := 11.95847;
   DATA[1161,30] := 1.724942;
   DATA[1161,31] := 1.302293;
   DATA[1161,32] := 0.7347566;
   DATA[1161,33] := 0.3084905;
   DATA[1161,34] := 2.0;
   DATA[1161,35] := 250.3525;
   DATA[1161,36] := 1.649953;
   DATA[1161,37] := 189.2944;
   DATA[1161,38] := 0.000128152;
   DATA[1161,39] := 1.0;
   DATA[1162,0] := 2.545239;
   DATA[1162,1] := 734.1051;
   DATA[1162,2] := 2.0;
   DATA[1162,3] := 1.0;
   DATA[1162,4] := 262.5288;
   DATA[1162,5] := 8.467573;
   DATA[1162,6] := 316.97;
   DATA[1162,8] := 1.0;
   DATA[1162,9] := 1.0;
   DATA[1162,10] := 1.0;
   DATA[1162,11] := 2.010372;
   DATA[1162,12] := 0.000256221;
   DATA[1162,13] := 1010.638;
   DATA[1162,14] := 1.0;
   DATA[1162,15] := 1.0;
   DATA[1162,16] := 1.0;
   DATA[1162,17] := 1.0;
   DATA[1162,18] := 1.0;
   DATA[1162,19] := 1.0;
   DATA[1162,20] := 148.808;
   DATA[1162,21] := 154.3963;
   DATA[1162,22] := 1.715567;
   DATA[1162,23] := 854.627;
   DATA[1162,24] := 2.0;
   DATA[1162,25] := 2.0;
   DATA[1162,26] := 7.87798;
   DATA[1162,27] := 143.6042;
   DATA[1162,28] := 263.0095;
   DATA[1162,29] := 11.95847;
   DATA[1162,30] := 1.724942;
   DATA[1162,31] := 1.305495;
   DATA[1162,32] := 0.7347566;
   DATA[1162,33] := 0.3084905;
   DATA[1162,34] := 2.0;
   DATA[1162,35] := 250.3525;
   DATA[1162,36] := 1.649953;
   DATA[1162,37] := 189.2464;
   DATA[1162,38] := 0.000128152;
   DATA[1162,39] := 1.0;
   DATA[1163,0] := 2.550684;
   DATA[1163,1] := 734.6154;
   DATA[1163,2] := 2.0;
   DATA[1163,3] := 1.0;
   DATA[1163,4] := 262.5288;
   DATA[1163,5] := 8.467573;
   DATA[1163,6] := 316.97;
   DATA[1163,8] := 1.0;
   DATA[1163,9] := 1.0;
   DATA[1163,10] := 1.0;
   DATA[1163,11] := 2.010372;
   DATA[1163,12] := 0.000256221;
   DATA[1163,13] := 1010.758;
   DATA[1163,14] := 1.0;
   DATA[1163,15] := 1.0;
   DATA[1163,16] := 1.0;
   DATA[1163,17] := 1.0;
   DATA[1163,18] := 1.0;
   DATA[1163,19] := 1.0;
   DATA[1163,20] := 148.808;
   DATA[1163,21] := 154.3963;
   DATA[1163,22] := 1.713645;
   DATA[1163,23] := 854.5501;
   DATA[1163,24] := 2.0;
   DATA[1163,25] := 2.0;
   DATA[1163,26] := 7.87798;
   DATA[1163,27] := 143.6042;
   DATA[1163,28] := 263.0095;
   DATA[1163,29] := 11.95847;
   DATA[1163,30] := 1.724942;
   DATA[1163,31] := 1.294607;
   DATA[1163,32] := 0.7347566;
   DATA[1163,33] := 0.3084905;
   DATA[1163,34] := 2.0;
   DATA[1163,35] := 250.3525;
   DATA[1163,36] := 1.649953;
   DATA[1163,37] := 189.1983;
   DATA[1163,38] := 0.000128152;
   DATA[1163,39] := 1.0;
   DATA[1164,0] := 2.550684;
   DATA[1164,1] := 735.2042;
   DATA[1164,2] := 2.0;
   DATA[1164,3] := 1.0;
   DATA[1164,4] := 262.5288;
   DATA[1164,5] := 8.467573;
   DATA[1164,6] := 316.97;
   DATA[1164,8] := 1.0;
   DATA[1164,9] := 1.0;
   DATA[1164,10] := 1.0;
   DATA[1164,11] := 2.010372;
   DATA[1164,12] := 0.000256221;
   DATA[1164,13] := 1010.839;
   DATA[1164,14] := 1.0;
   DATA[1164,15] := 1.0;
   DATA[1164,16] := 1.0;
   DATA[1164,17] := 1.0;
   DATA[1164,18] := 1.0;
   DATA[1164,19] := 1.0;
   DATA[1164,20] := 148.808;
   DATA[1164,21] := 154.5757;
   DATA[1164,22] := 1.713389;
   DATA[1164,23] := 854.3194;
   DATA[1164,24] := 2.0;
   DATA[1164,25] := 2.0;
   DATA[1164,26] := 7.87798;
   DATA[1164,27] := 143.6042;
   DATA[1164,28] := 263.0095;
   DATA[1164,29] := 11.95847;
   DATA[1164,30] := 1.724942;
   DATA[1164,31] := 1.283207;
   DATA[1164,32] := 0.7347566;
   DATA[1164,33] := 0.3084905;
   DATA[1164,34] := 2.0;
   DATA[1164,35] := 250.3525;
   DATA[1164,36] := 1.649953;
   DATA[1164,37] := 189.1022;
   DATA[1164,38] := 0.000128152;
   DATA[1164,39] := 1.0;
   DATA[1165,0] := 2.558691;
   DATA[1165,1] := 736.264;
   DATA[1165,2] := 2.0;
   DATA[1165,3] := 1.0;
   DATA[1165,4] := 262.5288;
   DATA[1165,5] := 8.467573;
   DATA[1165,6] := 316.97;
   DATA[1165,8] := 1.0;
   DATA[1165,9] := 1.0;
   DATA[1165,10] := 1.0;
   DATA[1165,11] := 2.010372;
   DATA[1165,12] := 0.000256221;
   DATA[1165,13] := 1010.959;
   DATA[1165,14] := 1.0;
   DATA[1165,15] := 1.0;
   DATA[1165,16] := 1.0;
   DATA[1165,17] := 1.0;
   DATA[1165,18] := 1.0;
   DATA[1165,19] := 1.0;
   DATA[1165,20] := 148.808;
   DATA[1165,21] := 154.6783;
   DATA[1165,22] := 1.713389;
   DATA[1165,23] := 854.2425;
   DATA[1165,24] := 2.0;
   DATA[1165,25] := 2.0;
   DATA[1165,26] := 7.87798;
   DATA[1165,27] := 143.6042;
   DATA[1165,28] := 263.0095;
   DATA[1165,29] := 11.95847;
   DATA[1165,30] := 1.724045;
   DATA[1165,31] := 1.287691;
   DATA[1165,32] := 0.7347566;
   DATA[1165,33] := 0.3084905;
   DATA[1165,34] := 2.0;
   DATA[1165,35] := 250.3525;
   DATA[1165,36] := 1.649953;
   DATA[1165,37] := 189.1022;
   DATA[1165,38] := 0.000128152;
   DATA[1165,39] := 1.0;
   DATA[1166,0] := 2.558691;
   DATA[1166,1] := 736.1855;
   DATA[1166,2] := 2.0;
   DATA[1166,3] := 1.0;
   DATA[1166,4] := 262.5288;
   DATA[1166,5] := 8.46533;
   DATA[1166,6] := 317.0982;
   DATA[1166,8] := 1.0;
   DATA[1166,9] := 1.0;
   DATA[1166,10] := 1.0;
   DATA[1166,11] := 2.010372;
   DATA[1166,12] := 0.000256221;
   DATA[1166,13] := 1010.919;
   DATA[1166,14] := 1.0;
   DATA[1166,15] := 1.0;
   DATA[1166,16] := 1.0;
   DATA[1166,17] := 1.0;
   DATA[1166,18] := 1.0;
   DATA[1166,19] := 1.0;
   DATA[1166,20] := 148.808;
   DATA[1166,21] := 154.6783;
   DATA[1166,22] := 1.71262;
   DATA[1166,23] := 854.0887;
   DATA[1166,24] := 2.0;
   DATA[1166,25] := 2.0;
   DATA[1166,26] := 7.87798;
   DATA[1166,27] := 143.6042;
   DATA[1166,28] := 263.0095;
   DATA[1166,29] := 11.95847;
   DATA[1166,30] := 1.724045;
   DATA[1166,31] := 1.282311;
   DATA[1166,32] := 0.7355248;
   DATA[1166,33] := 0.3084905;
   DATA[1166,34] := 2.0;
   DATA[1166,35] := 250.3525;
   DATA[1166,36] := 1.681991;
   DATA[1166,37] := 189.1022;
   DATA[1166,38] := 0.000128152;
   DATA[1166,39] := 1.0;
   DATA[1167,0] := 2.558691;
   DATA[1167,1] := 736.8528;
   DATA[1167,2] := 2.0;
   DATA[1167,3] := 1.0;
   DATA[1167,4] := 262.5288;
   DATA[1167,5] := 8.464369;
   DATA[1167,6] := 317.0982;
   DATA[1167,8] := 1.0;
   DATA[1167,9] := 1.0;
   DATA[1167,10] := 1.0;
   DATA[1167,11] := 2.010372;
   DATA[1167,12] := 0.000256221;
   DATA[1167,13] := 1010.879;
   DATA[1167,14] := 1.0;
   DATA[1167,15] := 1.0;
   DATA[1167,16] := 1.0;
   DATA[1167,17] := 1.0;
   DATA[1167,18] := 1.0;
   DATA[1167,19] := 1.0;
   DATA[1167,20] := 148.808;
   DATA[1167,21] := 154.6783;
   DATA[1167,22] := 1.713901;
   DATA[1167,23] := 853.4734;
   DATA[1167,24] := 2.0;
   DATA[1167,25] := 2.0;
   DATA[1167,26] := 7.87798;
   DATA[1167,27] := 143.6042;
   DATA[1167,28] := 263.0095;
   DATA[1167,29] := 11.95847;
   DATA[1167,30] := 1.724045;
   DATA[1167,31] := 1.281927;
   DATA[1167,32] := 0.7355248;
   DATA[1167,33] := 0.3084905;
   DATA[1167,34] := 2.0;
   DATA[1167,35] := 250.3525;
   DATA[1167,36] := 1.681991;
   DATA[1167,37] := 189.1022;
   DATA[1167,38] := 0.000128152;
   DATA[1167,39] := 1.0;
   DATA[1168,0] := 2.558691;
   DATA[1168,1] := 736.8528;
   DATA[1168,2] := 2.0;
   DATA[1168,3] := 1.0;
   DATA[1168,4] := 262.5288;
   DATA[1168,5] := 8.464369;
   DATA[1168,6] := 317.0982;
   DATA[1168,8] := 1.0;
   DATA[1168,9] := 1.0;
   DATA[1168,10] := 1.0;
   DATA[1168,11] := 2.010372;
   DATA[1168,12] := 0.000256221;
   DATA[1168,13] := 1010.758;
   DATA[1168,14] := 1.0;
   DATA[1168,15] := 1.0;
   DATA[1168,16] := 1.0;
   DATA[1168,17] := 1.0;
   DATA[1168,18] := 1.0;
   DATA[1168,19] := 1.0;
   DATA[1168,20] := 148.808;
   DATA[1168,21] := 154.627;
   DATA[1168,22] := 1.714029;
   DATA[1168,23] := 853.3196;
   DATA[1168,24] := 2.0;
   DATA[1168,25] := 2.0;
   DATA[1168,26] := 7.87798;
   DATA[1168,27] := 143.6042;
   DATA[1168,28] := 263.0095;
   DATA[1168,29] := 11.95847;
   DATA[1168,30] := 1.724045;
   DATA[1168,31] := 1.275522;
   DATA[1168,32] := 0.7355248;
   DATA[1168,33] := 0.3084905;
   DATA[1168,34] := 2.0;
   DATA[1168,35] := 250.3525;
   DATA[1168,36] := 1.681991;
   DATA[1168,37] := 189.1022;
   DATA[1168,38] := 0.000128152;
   DATA[1168,39] := 1.0;
   DATA[1169,0] := 2.558691;
   DATA[1169,1] := 737.1276;
   DATA[1169,2] := 2.0;
   DATA[1169,3] := 1.0;
   DATA[1169,4] := 262.5288;
   DATA[1169,5] := 8.464369;
   DATA[1169,6] := 317.0982;
   DATA[1169,8] := 1.0;
   DATA[1169,9] := 1.0;
   DATA[1169,10] := 1.0;
   DATA[1169,11] := 2.010372;
   DATA[1169,12] := 0.000256221;
   DATA[1169,13] := 1010.919;
   DATA[1169,14] := 1.0;
   DATA[1169,15] := 1.0;
   DATA[1169,16] := 1.0;
   DATA[1169,17] := 1.0;
   DATA[1169,18] := 1.0;
   DATA[1169,19] := 1.0;
   DATA[1169,20] := 148.808;
   DATA[1169,21] := 154.4476;
   DATA[1169,22] := 1.714029;
   DATA[1169,23] := 852.5506;
   DATA[1169,24] := 2.0;
   DATA[1169,25] := 2.0;
   DATA[1169,26] := 7.87798;
   DATA[1169,27] := 143.6042;
   DATA[1169,28] := 263.0095;
   DATA[1169,29] := 11.95847;
   DATA[1169,30] := 1.726993;
   DATA[1169,31] := 1.271679;
   DATA[1169,32] := 0.7355248;
   DATA[1169,33] := 0.3084905;
   DATA[1169,34] := 2.0;
   DATA[1169,35] := 250.3525;
   DATA[1169,36] := 1.681991;
   DATA[1169,37] := 189.1342;
   DATA[1169,38] := 0.000128152;
   DATA[1169,39] := 1.0;
   DATA[1170,0] := 2.551645;
   DATA[1170,1] := 737.4808;
   DATA[1170,2] := 2.0;
   DATA[1170,3] := 1.0;
   DATA[1170,4] := 262.5288;
   DATA[1170,5] := 8.464369;
   DATA[1170,6] := 317.0982;
   DATA[1170,8] := 1.0;
   DATA[1170,9] := 1.0;
   DATA[1170,10] := 1.0;
   DATA[1170,11] := 2.010372;
   DATA[1170,12] := 0.000256221;
   DATA[1170,13] := 1010.839;
   DATA[1170,14] := 1.0;
   DATA[1170,15] := 1.0;
   DATA[1170,16] := 1.0;
   DATA[1170,17] := 1.0;
   DATA[1170,18] := 1.0;
   DATA[1170,19] := 1.0;
   DATA[1170,20] := 148.808;
   DATA[1170,21] := 154.4476;
   DATA[1170,22] := 1.714029;
   DATA[1170,23] := 852.7429;
   DATA[1170,24] := 2.0;
   DATA[1170,25] := 2.0;
   DATA[1170,26] := 7.87798;
   DATA[1170,27] := 143.6042;
   DATA[1170,28] := 263.0095;
   DATA[1170,29] := 11.95847;
   DATA[1170,30] := 1.726993;
   DATA[1170,31] := 1.28641;
   DATA[1170,32] := 0.7355248;
   DATA[1170,33] := 0.3084905;
   DATA[1170,34] := 2.0;
   DATA[1170,35] := 250.3525;
   DATA[1170,36] := 1.681991;
   DATA[1170,37] := 189.2464;
   DATA[1170,38] := 0.000128152;
   DATA[1170,39] := 1.0;
   DATA[1171,0] := 2.540755;
   DATA[1171,1] := 737.6378;
   DATA[1171,2] := 2.0;
   DATA[1171,3] := 1.0;
   DATA[1171,4] := 262.5288;
   DATA[1171,5] := 8.464369;
   DATA[1171,6] := 317.0982;
   DATA[1171,8] := 1.0;
   DATA[1171,9] := 1.0;
   DATA[1171,10] := 1.0;
   DATA[1171,11] := 2.010372;
   DATA[1171,12] := 0.000256221;
   DATA[1171,13] := 1010.879;
   DATA[1171,14] := 1.0;
   DATA[1171,15] := 1.0;
   DATA[1171,16] := 1.0;
   DATA[1171,17] := 1.0;
   DATA[1171,18] := 1.0;
   DATA[1171,19] := 1.0;
   DATA[1171,20] := 148.808;
   DATA[1171,21] := 154.4476;
   DATA[1171,22] := 1.714029;
   DATA[1171,23] := 852.0123;
   DATA[1171,24] := 2.0;
   DATA[1171,25] := 2.0;
   DATA[1171,26] := 7.87798;
   DATA[1171,27] := 143.6042;
   DATA[1171,28] := 263.0095;
   DATA[1171,29] := 11.95847;
   DATA[1171,30] := 1.726993;
   DATA[1171,31] := 1.291789;
   DATA[1171,32] := 0.7355248;
   DATA[1171,33] := 0.3084905;
   DATA[1171,34] := 2.0;
   DATA[1171,35] := 250.3525;
   DATA[1171,36] := 1.681991;
   DATA[1171,37] := 189.2464;
   DATA[1171,38] := 0.000128152;
   DATA[1171,39] := 1.0;
   DATA[1172,0] := 2.539474;
   DATA[1172,1] := 739.0117;
   DATA[1172,2] := 2.0;
   DATA[1172,3] := 1.0;
   DATA[1172,4] := 262.5288;
   DATA[1172,5] := 8.464369;
   DATA[1172,6] := 317.0982;
   DATA[1172,8] := 1.0;
   DATA[1172,9] := 1.0;
   DATA[1172,10] := 1.0;
   DATA[1172,11] := 2.010372;
   DATA[1172,12] := 0.000256221;
   DATA[1172,13] := 1010.678;
   DATA[1172,14] := 1.0;
   DATA[1172,15] := 1.0;
   DATA[1172,16] := 1.0;
   DATA[1172,17] := 1.0;
   DATA[1172,18] := 1.0;
   DATA[1172,19] := 1.0;
   DATA[1172,20] := 148.808;
   DATA[1172,21] := 154.4476;
   DATA[1172,22] := 1.714029;
   DATA[1172,23] := 851.5894;
   DATA[1172,24] := 2.0;
   DATA[1172,25] := 2.0;
   DATA[1172,26] := 7.87798;
   DATA[1172,27] := 143.6042;
   DATA[1172,28] := 263.0095;
   DATA[1172,29] := 12.15073;
   DATA[1172,30] := 1.726993;
   DATA[1172,31] := 1.299603;
   DATA[1172,32] := 0.7355248;
   DATA[1172,33] := 0.3084905;
   DATA[1172,34] := 2.0;
   DATA[1172,35] := 250.3525;
   DATA[1172,36] := 1.681991;
   DATA[1172,37] := 189.2464;
   DATA[1172,38] := 0.000128152;
   DATA[1172,39] := 1.0;
   DATA[1173,0] := 2.536271;
   DATA[1173,1] := 739.522;
   DATA[1173,2] := 2.0;
   DATA[1173,3] := 1.0;
   DATA[1173,4] := 262.5288;
   DATA[1173,5] := 8.464369;
   DATA[1173,6] := 317.0982;
   DATA[1173,8] := 1.0;
   DATA[1173,9] := 1.0;
   DATA[1173,10] := 1.0;
   DATA[1173,11] := 2.010372;
   DATA[1173,12] := 0.000256221;
   DATA[1173,13] := 1010.758;
   DATA[1173,14] := 1.0;
   DATA[1173,15] := 1.0;
   DATA[1173,16] := 1.0;
   DATA[1173,17] := 1.0;
   DATA[1173,18] := 1.0;
   DATA[1173,19] := 1.0;
   DATA[1173,20] := 148.808;
   DATA[1173,21] := 154.4476;
   DATA[1173,22] := 1.715183;
   DATA[1173,23] := 851.1664;
   DATA[1173,24] := 2.0;
   DATA[1173,25] := 2.0;
   DATA[1173,26] := 7.87798;
   DATA[1173,27] := 143.6042;
   DATA[1173,28] := 263.0095;
   DATA[1173,29] := 12.15073;
   DATA[1173,30] := 1.726993;
   DATA[1173,31] := 1.302293;
   DATA[1173,32] := 0.7355248;
   DATA[1173,33] := 0.3084905;
   DATA[1173,34] := 2.0;
   DATA[1173,35] := 250.3525;
   DATA[1173,36] := 1.762086;
   DATA[1173,37] := 189.2464;
   DATA[1173,38] := 0.000128152;
   DATA[1173,39] := 1.0;
   DATA[1174,0] := 2.535631;
   DATA[1174,1] := 739.8752;
   DATA[1174,2] := 2.0;
   DATA[1174,3] := 1.0;
   DATA[1174,4] := 262.5288;
   DATA[1174,5] := 8.464369;
   DATA[1174,6] := 317.0982;
   DATA[1174,8] := 1.0;
   DATA[1174,9] := 1.0;
   DATA[1174,10] := 1.0;
   DATA[1174,11] := 2.010372;
   DATA[1174,12] := 0.000256221;
   DATA[1174,13] := 1010.638;
   DATA[1174,14] := 1.0;
   DATA[1174,15] := 1.0;
   DATA[1174,16] := 1.0;
   DATA[1174,17] := 1.0;
   DATA[1174,18] := 1.0;
   DATA[1174,19] := 1.0;
   DATA[1174,20] := 148.808;
   DATA[1174,21] := 154.4476;
   DATA[1174,22] := 1.715311;
   DATA[1174,23] := 850.8972;
   DATA[1174,24] := 2.0;
   DATA[1174,25] := 2.0;
   DATA[1174,26] := 7.87798;
   DATA[1174,27] := 143.6042;
   DATA[1174,28] := 263.0095;
   DATA[1174,29] := 12.15073;
   DATA[1174,30] := 1.726993;
   DATA[1174,31] := 1.30178;
   DATA[1174,32] := 0.7355248;
   DATA[1174,33] := 0.3084905;
   DATA[1174,34] := 2.0;
   DATA[1174,35] := 250.3525;
   DATA[1174,36] := 1.762086;
   DATA[1174,37] := 189.2464;
   DATA[1174,38] := 0.000128152;
   DATA[1174,39] := 1.0;
   DATA[1175,0] := 2.535631;
   DATA[1175,1] := 740.6995;
   DATA[1175,2] := 2.0;
   DATA[1175,3] := 1.0;
   DATA[1175,4] := 262.5288;
   DATA[1175,5] := 8.464369;
   DATA[1175,6] := 317.0982;
   DATA[1175,8] := 1.0;
   DATA[1175,9] := 1.0;
   DATA[1175,10] := 1.0;
   DATA[1175,11] := 2.010372;
   DATA[1175,12] := 0.000256221;
   DATA[1175,13] := 1010.919;
   DATA[1175,14] := 1.0;
   DATA[1175,15] := 1.0;
   DATA[1175,16] := 1.0;
   DATA[1175,17] := 1.0;
   DATA[1175,18] := 1.0;
   DATA[1175,19] := 1.0;
   DATA[1175,20] := 148.808;
   DATA[1175,21] := 154.4476;
   DATA[1175,22] := 1.716208;
   DATA[1175,23] := 850.4358;
   DATA[1175,24] := 2.0;
   DATA[1175,25] := 2.0;
   DATA[1175,26] := 7.87798;
   DATA[1175,27] := 143.6042;
   DATA[1175,28] := 263.0095;
   DATA[1175,29] := 12.15073;
   DATA[1175,30] := 1.726993;
   DATA[1175,31] := 1.291789;
   DATA[1175,32] := 0.7355248;
   DATA[1175,33] := 0.3084905;
   DATA[1175,34] := 2.0;
   DATA[1175,35] := 250.3525;
   DATA[1175,36] := 1.762086;
   DATA[1175,37] := 189.2464;
   DATA[1175,38] := 0.000128152;
   DATA[1175,39] := 1.0;
   DATA[1176,0] := 2.542036;
   DATA[1176,1] := 741.5631;
   DATA[1176,2] := 2.0;
   DATA[1176,3] := 1.0;
   DATA[1176,4] := 262.5288;
   DATA[1176,5] := 8.464369;
   DATA[1176,6] := 317.0982;
   DATA[1176,8] := 1.0;
   DATA[1176,9] := 1.0;
   DATA[1176,10] := 1.0;
   DATA[1176,11] := 2.010372;
   DATA[1176,12] := 0.000256221;
   DATA[1176,13] := 1010.839;
   DATA[1176,14] := 1.0;
   DATA[1176,15] := 1.0;
   DATA[1176,16] := 1.0;
   DATA[1176,17] := 1.0;
   DATA[1176,18] := 1.0;
   DATA[1176,19] := 1.0;
   DATA[1176,20] := 148.808;
   DATA[1176,21] := 154.4476;
   DATA[1176,22] := 1.717746;
   DATA[1176,23] := 850.3973;
   DATA[1176,24] := 2.0;
   DATA[1176,25] := 2.0;
   DATA[1176,26] := 7.87798;
   DATA[1176,27] := 143.6042;
   DATA[1176,28] := 263.0095;
   DATA[1176,29] := 12.07383;
   DATA[1176,30] := 1.725455;
   DATA[1176,31] := 1.296273;
   DATA[1176,32] := 0.7355248;
   DATA[1176,33] := 0.3084905;
   DATA[1176,34] := 2.0;
   DATA[1176,35] := 250.3525;
   DATA[1176,36] := 1.762086;
   DATA[1176,37] := 189.2464;
   DATA[1176,38] := 0.000128152;
   DATA[1176,39] := 1.0;
   DATA[1177,0] := 2.54684;
   DATA[1177,1] := 741.7593;
   DATA[1177,2] := 2.0;
   DATA[1177,3] := 1.0;
   DATA[1177,4] := 262.5288;
   DATA[1177,5] := 8.464369;
   DATA[1177,6] := 317.0982;
   DATA[1177,8] := 1.0;
   DATA[1177,9] := 1.0;
   DATA[1177,10] := 1.0;
   DATA[1177,11] := 2.010372;
   DATA[1177,12] := 0.000256221;
   DATA[1177,13] := 1010.638;
   DATA[1177,14] := 1.0;
   DATA[1177,15] := 1.0;
   DATA[1177,16] := 1.0;
   DATA[1177,17] := 1.0;
   DATA[1177,18] := 1.0;
   DATA[1177,19] := 1.0;
   DATA[1177,20] := 148.808;
   DATA[1177,21] := 154.4476;
   DATA[1177,22] := 1.717746;
   DATA[1177,23] := 850.2051;
   DATA[1177,24] := 2.0;
   DATA[1177,25] := 2.0;
   DATA[1177,26] := 7.87798;
   DATA[1177,27] := 143.6042;
   DATA[1177,28] := 263.0095;
   DATA[1177,29] := 12.07383;
   DATA[1177,30] := 1.725327;
   DATA[1177,31] := 1.3005;
   DATA[1177,32] := 0.7355248;
   DATA[1177,33] := 0.3084905;
   DATA[1177,34] := 2.0;
   DATA[1177,35] := 250.3525;
   DATA[1177,36] := 1.762086;
   DATA[1177,37] := 189.2464;
   DATA[1177,38] := 0.000128152;
   DATA[1177,39] := 1.0;
   DATA[1178,0] := 2.552285;
   DATA[1178,1] := 742.5052;
   DATA[1178,2] := 2.0;
   DATA[1178,3] := 1.0;
   DATA[1178,4] := 262.5288;
   DATA[1178,5] := 8.464369;
   DATA[1178,6] := 317.0982;
   DATA[1178,8] := 1.0;
   DATA[1178,9] := 1.0;
   DATA[1178,10] := 1.0;
   DATA[1178,11] := 2.010372;
   DATA[1178,12] := 0.000256221;
   DATA[1178,13] := 1010.919;
   DATA[1178,14] := 1.0;
   DATA[1178,15] := 1.0;
   DATA[1178,16] := 1.0;
   DATA[1178,17] := 1.0;
   DATA[1178,18] := 1.0;
   DATA[1178,19] := 1.0;
   DATA[1178,20] := 148.808;
   DATA[1178,21] := 154.4476;
   DATA[1178,22] := 1.717746;
   DATA[1178,23] := 850.2051;
   DATA[1178,24] := 2.0;
   DATA[1178,25] := 2.0;
   DATA[1178,26] := 7.87798;
   DATA[1178,27] := 143.6042;
   DATA[1178,28] := 263.0095;
   DATA[1178,29] := 12.07383;
   DATA[1178,30] := 1.724814;
   DATA[1178,31] := 1.286153;
   DATA[1178,32] := 0.7355248;
   DATA[1178,33] := 0.3084905;
   DATA[1178,34] := 2.0;
   DATA[1178,35] := 250.3525;
   DATA[1178,36] := 1.762086;
   DATA[1178,37] := 189.2464;
   DATA[1178,38] := 0.000128152;
   DATA[1178,39] := 1.0;
   DATA[1179,0] := 2.552285;
   DATA[1179,1] := 744.0753;
   DATA[1179,2] := 2.0;
   DATA[1179,3] := 1.0;
   DATA[1179,4] := 262.5288;
   DATA[1179,5] := 8.464369;
   DATA[1179,6] := 317.0982;
   DATA[1179,8] := 1.0;
   DATA[1179,9] := 1.0;
   DATA[1179,10] := 1.0;
   DATA[1179,11] := 2.010372;
   DATA[1179,12] := 0.000256221;
   DATA[1179,13] := 1010.758;
   DATA[1179,14] := 1.0;
   DATA[1179,15] := 1.0;
   DATA[1179,16] := 1.0;
   DATA[1179,17] := 1.0;
   DATA[1179,18] := 1.0;
   DATA[1179,19] := 1.0;
   DATA[1179,20] := 148.808;
   DATA[1179,21] := 154.4476;
   DATA[1179,22] := 1.717746;
   DATA[1179,23] := 849.7052;
   DATA[1179,24] := 2.0;
   DATA[1179,25] := 2.0;
   DATA[1179,26] := 7.87798;
   DATA[1179,27] := 143.6042;
   DATA[1179,28] := 263.0095;
   DATA[1179,29] := 12.07383;
   DATA[1179,30] := 1.724814;
   DATA[1179,31] := 1.263225;
   DATA[1179,32] := 0.7355248;
   DATA[1179,33] := 0.3084905;
   DATA[1179,34] := 2.0;
   DATA[1179,35] := 250.3525;
   DATA[1179,36] := 1.762086;
   DATA[1179,37] := 189.2464;
   DATA[1179,38] := 0.000128152;
   DATA[1179,39] := 1.0;
   DATA[1180,0] := 2.552285;
   DATA[1180,1] := 744.8604;
   DATA[1180,2] := 2.0;
   DATA[1180,3] := 1.0;
   DATA[1180,4] := 262.5288;
   DATA[1180,5] := 8.464369;
   DATA[1180,6] := 317.0982;
   DATA[1180,8] := 1.0;
   DATA[1180,9] := 1.0;
   DATA[1180,10] := 1.0;
   DATA[1180,11] := 2.010372;
   DATA[1180,12] := 0.000256221;
   DATA[1180,13] := 1010.919;
   DATA[1180,14] := 1.0;
   DATA[1180,15] := 1.0;
   DATA[1180,16] := 1.0;
   DATA[1180,17] := 1.0;
   DATA[1180,18] := 1.0;
   DATA[1180,19] := 1.0;
   DATA[1180,20] := 148.808;
   DATA[1180,21] := 154.4476;
   DATA[1180,22] := 1.717746;
   DATA[1180,23] := 849.859;
   DATA[1180,24] := 2.0;
   DATA[1180,25] := 2.0;
   DATA[1180,26] := 7.87798;
   DATA[1180,27] := 143.6042;
   DATA[1180,28] := 263.0095;
   DATA[1180,29] := 12.07383;
   DATA[1180,30] := 1.724814;
   DATA[1180,31] := 1.255284;
   DATA[1180,32] := 0.7355248;
   DATA[1180,33] := 0.3084905;
   DATA[1180,34] := 2.0;
   DATA[1180,35] := 250.3525;
   DATA[1180,36] := 1.762086;
   DATA[1180,37] := 189.2143;
   DATA[1180,38] := 0.000128152;
   DATA[1180,39] := 1.0;
   DATA[1181,0] := 2.550043;
   DATA[1181,1] := 745.1351;
   DATA[1181,2] := 2.0;
   DATA[1181,3] := 1.0;
   DATA[1181,4] := 262.5288;
   DATA[1181,5] := 8.464369;
   DATA[1181,6] := 317.0982;
   DATA[1181,8] := 1.0;
   DATA[1181,9] := 1.0;
   DATA[1181,10] := 1.0;
   DATA[1181,11] := 2.010372;
   DATA[1181,12] := 0.000256221;
   DATA[1181,13] := 1010.919;
   DATA[1181,14] := 1.0;
   DATA[1181,15] := 1.0;
   DATA[1181,16] := 1.0;
   DATA[1181,17] := 1.0;
   DATA[1181,18] := 1.0;
   DATA[1181,19] := 1.0;
   DATA[1181,20] := 148.808;
   DATA[1181,21] := 154.4476;
   DATA[1181,22] := 1.717746;
   DATA[1181,23] := 849.3591;
   DATA[1181,24] := 2.0;
   DATA[1181,25] := 2.0;
   DATA[1181,26] := 7.87798;
   DATA[1181,27] := 143.6042;
   DATA[1181,28] := 263.0095;
   DATA[1181,29] := 12.07383;
   DATA[1181,30] := 1.725327;
   DATA[1181,31] := 1.260535;
   DATA[1181,32] := 0.7355248;
   DATA[1181,33] := 0.3084905;
   DATA[1181,34] := 2.0;
   DATA[1181,35] := 250.3525;
   DATA[1181,36] := 1.762086;
   DATA[1181,37] := 189.1662;
   DATA[1181,38] := 0.000128152;
   DATA[1181,39] := 1.0;
   DATA[1182,0] := 2.54652;
   DATA[1182,1] := 745.6454;
   DATA[1182,2] := 2.0;
   DATA[1182,3] := 1.0;
   DATA[1182,4] := 262.5288;
   DATA[1182,5] := 8.464369;
   DATA[1182,6] := 317.0982;
   DATA[1182,8] := 1.0;
   DATA[1182,9] := 1.0;
   DATA[1182,10] := 1.0;
   DATA[1182,11] := 2.010372;
   DATA[1182,12] := 0.000256221;
   DATA[1182,13] := 1011.119;
   DATA[1182,14] := 1.0;
   DATA[1182,15] := 1.0;
   DATA[1182,16] := 1.0;
   DATA[1182,17] := 1.0;
   DATA[1182,18] := 1.0;
   DATA[1182,19] := 1.0;
   DATA[1182,20] := 148.808;
   DATA[1182,21] := 154.4476;
   DATA[1182,22] := 1.717746;
   DATA[1182,23] := 848.8977;
   DATA[1182,24] := 2.0;
   DATA[1182,25] := 2.0;
   DATA[1182,26] := 7.87798;
   DATA[1182,27] := 143.6042;
   DATA[1182,28] := 263.0095;
   DATA[1182,29] := 12.07383;
   DATA[1182,30] := 1.726609;
   DATA[1182,31] := 1.274881;
   DATA[1182,32] := 0.7355248;
   DATA[1182,33] := 0.3084905;
   DATA[1182,34] := 2.0;
   DATA[1182,35] := 250.3525;
   DATA[1182,36] := 1.762086;
   DATA[1182,37] := 189.0381;
   DATA[1182,38] := 0.000128152;
   DATA[1182,39] := 1.0;
   DATA[1183,0] := 2.54652;
   DATA[1183,1] := 746.1557;
   DATA[1183,2] := 2.0;
   DATA[1183,3] := 1.0;
   DATA[1183,4] := 262.5288;
   DATA[1183,5] := 8.464369;
   DATA[1183,6] := 317.0982;
   DATA[1183,8] := 1.0;
   DATA[1183,9] := 1.0;
   DATA[1183,10] := 1.0;
   DATA[1183,11] := 2.010372;
   DATA[1183,12] := 0.000256221;
   DATA[1183,13] := 1011.159;
   DATA[1183,14] := 1.0;
   DATA[1183,15] := 1.0;
   DATA[1183,16] := 1.0;
   DATA[1183,17] := 1.0;
   DATA[1183,18] := 1.0;
   DATA[1183,19] := 1.0;
   DATA[1183,20] := 148.808;
   DATA[1183,21] := 154.4476;
   DATA[1183,22] := 1.717746;
   DATA[1183,23] := 847.7826;
   DATA[1183,24] := 2.0;
   DATA[1183,25] := 2.0;
   DATA[1183,26] := 7.87798;
   DATA[1183,27] := 143.6042;
   DATA[1183,28] := 263.0095;
   DATA[1183,29] := 12.07383;
   DATA[1183,30] := 1.726609;
   DATA[1183,31] := 1.298834;
   DATA[1183,32] := 0.7352687;
   DATA[1183,33] := 0.3084905;
   DATA[1183,34] := 2.0;
   DATA[1183,35] := 250.3525;
   DATA[1183,36] := 1.617916;
   DATA[1183,37] := 189.0381;
   DATA[1183,38] := 0.000128152;
   DATA[1183,39] := 1.0;
   DATA[1184,0] := 2.542036;
   DATA[1184,1] := 746.666;
   DATA[1184,2] := 2.0;
   DATA[1184,3] := 1.0;
   DATA[1184,4] := 262.5288;
   DATA[1184,5] := 8.464369;
   DATA[1184,6] := 317.0982;
   DATA[1184,8] := 1.0;
   DATA[1184,9] := 1.0;
   DATA[1184,10] := 1.0;
   DATA[1184,11] := 2.010372;
   DATA[1184,12] := 0.000256221;
   DATA[1184,13] := 1011.159;
   DATA[1184,14] := 1.0;
   DATA[1184,15] := 1.0;
   DATA[1184,16] := 1.0;
   DATA[1184,17] := 1.0;
   DATA[1184,18] := 1.0;
   DATA[1184,19] := 1.0;
   DATA[1184,20] := 148.808;
   DATA[1184,21] := 154.4476;
   DATA[1184,22] := 1.717746;
   DATA[1184,23] := 847.5519;
   DATA[1184,24] := 2.0;
   DATA[1184,25] := 2.0;
   DATA[1184,26] := 7.87798;
   DATA[1184,27] := 143.5786;
   DATA[1184,28] := 263.0095;
   DATA[1184,29] := 12.07383;
   DATA[1184,30] := 1.726609;
   DATA[1184,31] := 1.302165;
   DATA[1184,32] := 0.7352687;
   DATA[1184,33] := 0.3084905;
   DATA[1184,34] := 2.0;
   DATA[1184,35] := 250.3525;
   DATA[1184,36] := 1.617916;
   DATA[1184,37] := 189.0381;
   DATA[1184,38] := 0.000128152;
   DATA[1184,39] := 1.0;
   DATA[1185,0] := 2.539474;
   DATA[1185,1] := 746.823;
   DATA[1185,2] := 2.0;
   DATA[1185,3] := 1.0;
   DATA[1185,4] := 262.5288;
   DATA[1185,5] := 8.464369;
   DATA[1185,6] := 317.0982;
   DATA[1185,8] := 1.0;
   DATA[1185,9] := 1.0;
   DATA[1185,10] := 1.0;
   DATA[1185,11] := 2.010372;
   DATA[1185,12] := 0.000256221;
   DATA[1185,13] := 1011.239;
   DATA[1185,14] := 1.0;
   DATA[1185,15] := 1.0;
   DATA[1185,16] := 1.0;
   DATA[1185,17] := 1.0;
   DATA[1185,18] := 1.0;
   DATA[1185,19] := 1.0;
   DATA[1185,20] := 148.808;
   DATA[1185,21] := 154.4476;
   DATA[1185,22] := 1.717746;
   DATA[1185,23] := 847.2443;
   DATA[1185,24] := 2.0;
   DATA[1185,25] := 2.0;
   DATA[1185,26] := 7.87798;
   DATA[1185,27] := 143.5786;
   DATA[1185,28] := 263.0095;
   DATA[1185,29] := 12.07383;
   DATA[1185,30] := 1.726609;
   DATA[1185,31] := 1.290124;
   DATA[1185,32] := 0.7352687;
   DATA[1185,33] := 0.3084905;
   DATA[1185,34] := 2.0;
   DATA[1185,35] := 250.3525;
   DATA[1185,36] := 1.617916;
   DATA[1185,37] := 189.0381;
   DATA[1185,38] := 0.000128152;
   DATA[1185,39] := 1.0;
   DATA[1186,0] := 2.539474;
   DATA[1186,1] := 747.5295;
   DATA[1186,2] := 2.0;
   DATA[1186,3] := 1.0;
   DATA[1186,4] := 262.5288;
   DATA[1186,5] := 8.464369;
   DATA[1186,6] := 317.0982;
   DATA[1186,8] := 1.0;
   DATA[1186,9] := 1.0;
   DATA[1186,10] := 1.0;
   DATA[1186,11] := 2.010372;
   DATA[1186,12] := 0.000256221;
   DATA[1186,13] := 1011.039;
   DATA[1186,14] := 1.0;
   DATA[1186,15] := 1.0;
   DATA[1186,16] := 1.0;
   DATA[1186,17] := 1.0;
   DATA[1186,18] := 1.0;
   DATA[1186,19] := 1.0;
   DATA[1186,20] := 148.808;
   DATA[1186,21] := 154.4476;
   DATA[1186,22] := 1.717746;
   DATA[1186,23] := 847.1674;
   DATA[1186,24] := 2.0;
   DATA[1186,25] := 2.0;
   DATA[1186,26] := 7.87798;
   DATA[1186,27] := 143.5786;
   DATA[1186,28] := 263.0095;
   DATA[1186,29] := 12.07383;
   DATA[1186,30] := 1.726609;
   DATA[1186,31] := 1.277699;
   DATA[1186,32] := 0.7352687;
   DATA[1186,33] := 0.3084905;
   DATA[1186,34] := 2.0;
   DATA[1186,35] := 250.3525;
   DATA[1186,36] := 1.617916;
   DATA[1186,37] := 189.2143;
   DATA[1186,38] := 0.000128152;
   DATA[1186,39] := 1.0;
   DATA[1187,0] := 2.545559;
   DATA[1187,1] := 748.0005;
   DATA[1187,2] := 2.0;
   DATA[1187,3] := 1.0;
   DATA[1187,4] := 262.5288;
   DATA[1187,5] := 8.464369;
   DATA[1187,6] := 317.0982;
   DATA[1187,8] := 1.0;
   DATA[1187,9] := 1.0;
   DATA[1187,10] := 1.0;
   DATA[1187,11] := 2.010372;
   DATA[1187,12] := 0.000256221;
   DATA[1187,13] := 1011.159;
   DATA[1187,14] := 1.0;
   DATA[1187,15] := 1.0;
   DATA[1187,16] := 1.0;
   DATA[1187,17] := 1.0;
   DATA[1187,18] := 1.0;
   DATA[1187,19] := 1.0;
   DATA[1187,20] := 148.808;
   DATA[1187,21] := 154.4476;
   DATA[1187,22] := 1.717746;
   DATA[1187,23] := 846.9367;
   DATA[1187,24] := 2.0;
   DATA[1187,25] := 2.0;
   DATA[1187,26] := 7.87798;
   DATA[1187,27] := 143.5786;
   DATA[1187,28] := 263.0095;
   DATA[1187,29] := 12.07383;
   DATA[1187,30] := 1.726609;
   DATA[1187,31] := 1.27232;
   DATA[1187,32] := 0.7352687;
   DATA[1187,33] := 0.3084905;
   DATA[1187,34] := 2.0;
   DATA[1187,35] := 250.3525;
   DATA[1187,36] := 1.617916;
   DATA[1187,37] := 189.2784;
   DATA[1187,38] := 0.000128152;
   DATA[1187,39] := 1.0;
   DATA[1188,0] := 2.552285;
   DATA[1188,1] := 747.8436;
   DATA[1188,2] := 2.0;
   DATA[1188,3] := 1.0;
   DATA[1188,4] := 262.5288;
   DATA[1188,5] := 8.464369;
   DATA[1188,6] := 317.0982;
   DATA[1188,8] := 1.0;
   DATA[1188,9] := 1.0;
   DATA[1188,10] := 1.0;
   DATA[1188,11] := 2.010372;
   DATA[1188,12] := 0.000256221;
   DATA[1188,13] := 1011.039;
   DATA[1188,14] := 1.0;
   DATA[1188,15] := 1.0;
   DATA[1188,16] := 1.0;
   DATA[1188,17] := 1.0;
   DATA[1188,18] := 1.0;
   DATA[1188,19] := 1.0;
   DATA[1188,20] := 148.808;
   DATA[1188,21] := 154.4476;
   DATA[1188,22] := 1.717746;
   DATA[1188,23] := 846.3984;
   DATA[1188,24] := 2.0;
   DATA[1188,25] := 2.0;
   DATA[1188,26] := 7.87798;
   DATA[1188,27] := 143.5786;
   DATA[1188,28] := 263.0095;
   DATA[1188,29] := 12.07383;
   DATA[1188,30] := 1.726609;
   DATA[1188,31] := 1.282439;
   DATA[1188,32] := 0.7352687;
   DATA[1188,33] := 0.3084905;
   DATA[1188,34] := 2.0;
   DATA[1188,35] := 250.3525;
   DATA[1188,36] := 1.617916;
   DATA[1188,37] := 189.2784;
   DATA[1188,38] := 0.000128152;
   DATA[1188,39] := 1.0;
   DATA[1189,0] := 2.556129;
   DATA[1189,1] := 747.8043;
   DATA[1189,2] := 2.0;
   DATA[1189,3] := 1.0;
   DATA[1189,4] := 262.5288;
   DATA[1189,5] := 8.464369;
   DATA[1189,6] := 317.0982;
   DATA[1189,8] := 1.0;
   DATA[1189,9] := 1.0;
   DATA[1189,10] := 1.0;
   DATA[1189,11] := 2.010372;
   DATA[1189,12] := 0.000256221;
   DATA[1189,13] := 1011.119;
   DATA[1189,14] := 1.0;
   DATA[1189,15] := 1.0;
   DATA[1189,16] := 1.0;
   DATA[1189,17] := 1.0;
   DATA[1189,18] := 1.0;
   DATA[1189,19] := 1.0;
   DATA[1189,20] := 148.808;
   DATA[1189,21] := 154.4476;
   DATA[1189,22] := 1.717746;
   DATA[1189,23] := 846.0139;
   DATA[1189,24] := 2.0;
   DATA[1189,25] := 2.0;
   DATA[1189,26] := 7.87798;
   DATA[1189,27] := 143.5786;
   DATA[1189,28] := 263.0095;
   DATA[1189,29] := 12.07383;
   DATA[1189,30] := 1.723532;
   DATA[1189,31] := 1.297041;
   DATA[1189,32] := 0.7352687;
   DATA[1189,33] := 0.3084905;
   DATA[1189,34] := 2.0;
   DATA[1189,35] := 250.3525;
   DATA[1189,36] := 1.617916;
   DATA[1189,37] := 189.2784;
   DATA[1189,38] := 0.000128152;
   DATA[1189,39] := 1.0;
   DATA[1190,0] := 2.557089;
   DATA[1190,1] := 748.3146;
   DATA[1190,2] := 2.0;
   DATA[1190,3] := 1.0;
   DATA[1190,4] := 262.5288;
   DATA[1190,5] := 8.464369;
   DATA[1190,6] := 317.0982;
   DATA[1190,8] := 1.0;
   DATA[1190,9] := 1.0;
   DATA[1190,10] := 1.0;
   DATA[1190,11] := 2.010372;
   DATA[1190,12] := 0.000256221;
   DATA[1190,13] := 1010.879;
   DATA[1190,14] := 1.0;
   DATA[1190,15] := 1.0;
   DATA[1190,16] := 1.0;
   DATA[1190,17] := 1.0;
   DATA[1190,18] := 1.0;
   DATA[1190,19] := 1.0;
   DATA[1190,20] := 148.808;
   DATA[1190,21] := 154.4988;
   DATA[1190,22] := 1.717489;
   DATA[1190,23] := 845.7831;
   DATA[1190,24] := 2.0;
   DATA[1190,25] := 2.0;
   DATA[1190,26] := 7.87798;
   DATA[1190,27] := 143.5786;
   DATA[1190,28] := 263.0095;
   DATA[1190,29] := 12.07383;
   DATA[1190,30] := 1.723532;
   DATA[1190,31] := 1.296273;
   DATA[1190,32] := 0.7352687;
   DATA[1190,33] := 0.3084905;
   DATA[1190,34] := 2.0;
   DATA[1190,35] := 250.3525;
   DATA[1190,36] := 1.617916;
   DATA[1190,37] := 189.2464;
   DATA[1190,38] := 0.000128152;
   DATA[1190,39] := 1.0;
   DATA[1191,0] := 2.557089;
   DATA[1191,1] := 748.4716;
   DATA[1191,2] := 2.0;
   DATA[1191,3] := 1.0;
   DATA[1191,4] := 262.5288;
   DATA[1191,5] := 8.464369;
   DATA[1191,6] := 317.0982;
   DATA[1191,8] := 1.0;
   DATA[1191,9] := 1.0;
   DATA[1191,10] := 1.0;
   DATA[1191,11] := 2.010372;
   DATA[1191,12] := 0.000256221;
   DATA[1191,13] := 1011.039;
   DATA[1191,14] := 1.0;
   DATA[1191,15] := 1.0;
   DATA[1191,16] := 1.0;
   DATA[1191,17] := 1.0;
   DATA[1191,18] := 1.0;
   DATA[1191,19] := 1.0;
   DATA[1191,20] := 148.808;
   DATA[1191,21] := 154.5501;
   DATA[1191,22] := 1.717105;
   DATA[1191,23] := 844.8987;
   DATA[1191,24] := 2.0;
   DATA[1191,25] := 2.0;
   DATA[1191,26] := 7.87798;
   DATA[1191,27] := 143.5786;
   DATA[1191,28] := 263.0095;
   DATA[1191,29] := 12.07383;
   DATA[1191,30] := 1.723532;
   DATA[1191,31] := 1.296529;
   DATA[1191,32] := 0.7352687;
   DATA[1191,33] := 0.3084905;
   DATA[1191,34] := 2.0;
   DATA[1191,35] := 250.3525;
   DATA[1191,36] := 1.665972;
   DATA[1191,37] := 189.1022;
   DATA[1191,38] := 0.000128152;
   DATA[1191,39] := 1.0;
   DATA[1192,0] := 2.556129;
   DATA[1192,1] := 748.7856;
   DATA[1192,2] := 2.0;
   DATA[1192,3] := 1.0;
   DATA[1192,4] := 262.5288;
   DATA[1192,5] := 8.464369;
   DATA[1192,6] := 317.0982;
   DATA[1192,8] := 1.0;
   DATA[1192,9] := 1.0;
   DATA[1192,10] := 1.0;
   DATA[1192,11] := 2.010372;
   DATA[1192,12] := 0.000256221;
   DATA[1192,13] := 1010.758;
   DATA[1192,14] := 1.0;
   DATA[1192,15] := 1.0;
   DATA[1192,16] := 1.0;
   DATA[1192,17] := 1.0;
   DATA[1192,18] := 1.0;
   DATA[1192,19] := 1.0;
   DATA[1192,20] := 148.808;
   DATA[1192,21] := 154.5501;
   DATA[1192,22] := 1.717105;
   DATA[1192,23] := 844.6296;
   DATA[1192,24] := 2.0;
   DATA[1192,25] := 2.0;
   DATA[1192,26] := 7.87798;
   DATA[1192,27] := 143.5786;
   DATA[1192,28] := 263.0095;
   DATA[1192,29] := 12.07383;
   DATA[1192,30] := 1.725968;
   DATA[1192,31] := 1.286282;
   DATA[1192,32] := 0.7352687;
   DATA[1192,33] := 0.3084905;
   DATA[1192,34] := 2.0;
   DATA[1192,35] := 250.2243;
   DATA[1192,36] := 1.665972;
   DATA[1192,37] := 189.1022;
   DATA[1192,38] := 0.000128152;
   DATA[1192,39] := 1.0;
   DATA[1193,0] := 2.551965;
   DATA[1193,1] := 749.8062;
   DATA[1193,2] := 2.0;
   DATA[1193,3] := 1.0;
   DATA[1193,4] := 262.5288;
   DATA[1193,5] := 8.464369;
   DATA[1193,6] := 317.0982;
   DATA[1193,8] := 1.0;
   DATA[1193,9] := 1.0;
   DATA[1193,10] := 1.0;
   DATA[1193,11] := 2.010372;
   DATA[1193,12] := 0.000256221;
   DATA[1193,13] := 1010.959;
   DATA[1193,14] := 1.0;
   DATA[1193,15] := 1.0;
   DATA[1193,16] := 1.0;
   DATA[1193,17] := 1.0;
   DATA[1193,18] := 1.0;
   DATA[1193,19] := 1.0;
   DATA[1193,20] := 148.808;
   DATA[1193,21] := 154.5501;
   DATA[1193,22] := 1.715952;
   DATA[1193,23] := 844.1682;
   DATA[1193,24] := 2.0;
   DATA[1193,25] := 2.0;
   DATA[1193,26] := 7.87798;
   DATA[1193,27] := 143.5786;
   DATA[1193,28] := 263.0095;
   DATA[1193,29] := 12.07383;
   DATA[1193,30] := 1.725968;
   DATA[1193,31] := 1.272064;
   DATA[1193,32] := 0.7352687;
   DATA[1193,33] := 0.3084905;
   DATA[1193,34] := 2.0;
   DATA[1193,35] := 250.2243;
   DATA[1193,36] := 1.665972;
   DATA[1193,37] := 189.1022;
   DATA[1193,38] := 0.000128152;
   DATA[1193,39] := 1.0;
   DATA[1194,0] := 2.54652;
   DATA[1194,1] := 749.7669;
   DATA[1194,2] := 2.0;
   DATA[1194,3] := 1.0;
   DATA[1194,4] := 262.5288;
   DATA[1194,5] := 8.464369;
   DATA[1194,6] := 317.0982;
   DATA[1194,8] := 1.0;
   DATA[1194,9] := 1.0;
   DATA[1194,10] := 1.0;
   DATA[1194,11] := 2.010372;
   DATA[1194,12] := 0.000256221;
   DATA[1194,13] := 1010.879;
   DATA[1194,14] := 1.0;
   DATA[1194,15] := 1.0;
   DATA[1194,16] := 1.0;
   DATA[1194,17] := 1.0;
   DATA[1194,18] := 1.0;
   DATA[1194,19] := 1.0;
   DATA[1194,20] := 148.808;
   DATA[1194,21] := 154.5501;
   DATA[1194,22] := 1.715439;
   DATA[1194,23] := 843.9374;
   DATA[1194,24] := 2.0;
   DATA[1194,25] := 2.0;
   DATA[1194,26] := 7.87798;
   DATA[1194,27] := 143.5786;
   DATA[1194,28] := 263.0095;
   DATA[1194,29] := 12.07383;
   DATA[1194,30] := 1.725968;
   DATA[1194,31] := 1.267452;
   DATA[1194,32] := 0.7352687;
   DATA[1194,33] := 0.3084905;
   DATA[1194,34] := 2.0;
   DATA[1194,35] := 250.2243;
   DATA[1194,36] := 1.665972;
   DATA[1194,37] := 189.1022;
   DATA[1194,38] := 0.000128152;
   DATA[1194,39] := 1.0;
   DATA[1195,0] := 2.542356;
   DATA[1195,1] := 750.0809;
   DATA[1195,2] := 2.0;
   DATA[1195,3] := 1.0;
   DATA[1195,4] := 262.5288;
   DATA[1195,5] := 8.464369;
   DATA[1195,6] := 317.0982;
   DATA[1195,8] := 1.0;
   DATA[1195,9] := 1.0;
   DATA[1195,10] := 1.0;
   DATA[1195,11] := 2.010372;
   DATA[1195,12] := 0.000256221;
   DATA[1195,13] := 1011.039;
   DATA[1195,14] := 1.0;
   DATA[1195,15] := 1.0;
   DATA[1195,16] := 1.0;
   DATA[1195,17] := 1.0;
   DATA[1195,18] := 1.0;
   DATA[1195,19] := 1.0;
   DATA[1195,20] := 148.808;
   DATA[1195,21] := 154.5501;
   DATA[1195,22] := 1.715439;
   DATA[1195,23] := 843.3991;
   DATA[1195,24] := 2.0;
   DATA[1195,25] := 2.0;
   DATA[1195,26] := 7.87798;
   DATA[1195,27] := 143.5786;
   DATA[1195,28] := 263.0095;
   DATA[1195,29] := 12.07383;
   DATA[1195,30] := 1.725968;
   DATA[1195,31] := 1.261304;
   DATA[1195,32] := 0.7352687;
   DATA[1195,33] := 0.3084905;
   DATA[1195,34] := 2.0;
   DATA[1195,35] := 250.2243;
   DATA[1195,36] := 1.665972;
   DATA[1195,37] := 189.1983;
   DATA[1195,38] := 0.000128152;
   DATA[1195,39] := 1.0;
   DATA[1196,0] := 2.535951;
   DATA[1196,1] := 750.4735;
   DATA[1196,2] := 2.0;
   DATA[1196,3] := 1.0;
   DATA[1196,4] := 262.5288;
   DATA[1196,5] := 8.464369;
   DATA[1196,6] := 317.0982;
   DATA[1196,8] := 1.0;
   DATA[1196,9] := 1.0;
   DATA[1196,10] := 1.0;
   DATA[1196,11] := 2.010372;
   DATA[1196,12] := 0.000256221;
   DATA[1196,13] := 1010.919;
   DATA[1196,14] := 1.0;
   DATA[1196,15] := 1.0;
   DATA[1196,16] := 1.0;
   DATA[1196,17] := 1.0;
   DATA[1196,18] := 1.0;
   DATA[1196,19] := 1.0;
   DATA[1196,20] := 148.808;
   DATA[1196,21] := 154.5501;
   DATA[1196,22] := 1.715439;
   DATA[1196,23] := 843.0915;
   DATA[1196,24] := 2.0;
   DATA[1196,25] := 2.0;
   DATA[1196,26] := 7.87798;
   DATA[1196,27] := 143.5786;
   DATA[1196,28] := 263.0095;
   DATA[1196,29] := 12.07383;
   DATA[1196,30] := 1.725968;
   DATA[1196,31] := 1.25823;
   DATA[1196,32] := 0.7352687;
   DATA[1196,33] := 0.3084905;
   DATA[1196,34] := 2.0;
   DATA[1196,35] := 250.4326;
   DATA[1196,36] := 1.69801;
   DATA[1196,37] := 189.1983;
   DATA[1196,38] := 0.000128152;
   DATA[1196,39] := 1.0;
   DATA[1197,0] := 2.535951;
   DATA[1197,1] := 751.1407;
   DATA[1197,2] := 2.0;
   DATA[1197,3] := 1.0;
   DATA[1197,4] := 262.5288;
   DATA[1197,5] := 8.464369;
   DATA[1197,6] := 317.0982;
   DATA[1197,8] := 1.0;
   DATA[1197,9] := 1.0;
   DATA[1197,10] := 1.0;
   DATA[1197,11] := 2.010372;
   DATA[1197,12] := 0.000256221;
   DATA[1197,13] := 1011.079;
   DATA[1197,14] := 1.0;
   DATA[1197,15] := 1.0;
   DATA[1197,16] := 1.0;
   DATA[1197,17] := 1.0;
   DATA[1197,18] := 1.0;
   DATA[1197,19] := 1.0;
   DATA[1197,20] := 148.808;
   DATA[1197,21] := 154.5501;
   DATA[1197,22] := 1.715439;
   DATA[1197,23] := 842.5916;
   DATA[1197,24] := 2.0;
   DATA[1197,25] := 2.0;
   DATA[1197,26] := 7.87798;
   DATA[1197,27] := 143.5786;
   DATA[1197,28] := 263.0095;
   DATA[1197,29] := 12.07383;
   DATA[1197,30] := 1.725968;
   DATA[1197,31] := 1.248495;
   DATA[1197,32] := 0.7352687;
   DATA[1197,33] := 0.3084905;
   DATA[1197,34] := 2.0;
   DATA[1197,35] := 250.4326;
   DATA[1197,36] := 1.69801;
   DATA[1197,37] := 189.1983;
   DATA[1197,38] := 0.000128152;
   DATA[1197,39] := 1.0;
   DATA[1198,0] := 2.535951;
   DATA[1198,1] := 751.7688;
   DATA[1198,2] := 2.0;
   DATA[1198,3] := 1.0;
   DATA[1198,4] := 262.5288;
   DATA[1198,5] := 8.464369;
   DATA[1198,6] := 317.0982;
   DATA[1198,8] := 1.0;
   DATA[1198,9] := 1.0;
   DATA[1198,10] := 1.0;
   DATA[1198,11] := 2.010372;
   DATA[1198,12] := 0.000256221;
   DATA[1198,13] := 1010.678;
   DATA[1198,14] := 1.0;
   DATA[1198,15] := 1.0;
   DATA[1198,16] := 1.0;
   DATA[1198,17] := 1.0;
   DATA[1198,18] := 1.0;
   DATA[1198,19] := 1.0;
   DATA[1198,20] := 148.808;
   DATA[1198,21] := 154.5501;
   DATA[1198,22] := 1.715439;
   DATA[1198,23] := 842.1687;
   DATA[1198,24] := 2.0;
   DATA[1198,25] := 2.0;
   DATA[1198,26] := 7.87798;
   DATA[1198,27] := 143.5786;
   DATA[1198,28] := 263.0095;
   DATA[1198,29] := 12.07383;
   DATA[1198,30] := 1.725968;
   DATA[1198,31] := 1.245293;
   DATA[1198,32] := 0.7352687;
   DATA[1198,33] := 0.3070813;
   DATA[1198,34] := 2.0;
   DATA[1198,35] := 250.4326;
   DATA[1198,36] := 1.69801;
   DATA[1198,37] := 189.1983;
   DATA[1198,38] := 0.000128152;
   DATA[1198,39] := 1.0;
   DATA[1199,0] := 2.542356;
   DATA[1199,1] := 752.3184;
   DATA[1199,2] := 2.0;
   DATA[1199,3] := 1.0;
   DATA[1199,4] := 262.5288;
   DATA[1199,5] := 8.464369;
   DATA[1199,6] := 317.0982;
   DATA[1199,8] := 1.0;
   DATA[1199,9] := 1.0;
   DATA[1199,10] := 1.0;
   DATA[1199,11] := 2.010372;
   DATA[1199,12] := 0.000256221;
   DATA[1199,13] := 1010.959;
   DATA[1199,14] := 1.0;
   DATA[1199,15] := 1.0;
   DATA[1199,16] := 1.0;
   DATA[1199,17] := 1.0;
   DATA[1199,18] := 1.0;
   DATA[1199,19] := 1.0;
   DATA[1199,20] := 148.808;
   DATA[1199,21] := 154.5501;
   DATA[1199,22] := 1.715439;
   DATA[1199,23] := 841.8226;
   DATA[1199,24] := 2.0;
   DATA[1199,25] := 2.0;
   DATA[1199,26] := 7.87798;
   DATA[1199,27] := 143.5786;
   DATA[1199,28] := 263.0095;
   DATA[1199,29] := 12.07383;
   DATA[1199,30] := 1.725968;
   DATA[1199,31] := 1.253619;
   DATA[1199,32] := 0.7352687;
   DATA[1199,33] := 0.3070813;
   DATA[1199,34] := 2.0;
   DATA[1199,35] := 250.4326;
   DATA[1199,36] := 1.69801;
   DATA[1199,37] := 189.1983;
   DATA[1199,38] := 0.000128152;
   DATA[1199,39] := 1.0;
   DATA[1200,0] := 2.542356;
   DATA[1200,1] := 752.3184;
   DATA[1200,2] := 2.0;
   DATA[1200,3] := 1.0;
   DATA[1200,4] := 262.5288;
   DATA[1200,5] := 8.464369;
   DATA[1200,6] := 317.0982;
   DATA[1200,8] := 1.0;
   DATA[1200,9] := 1.0;
   DATA[1200,10] := 1.0;
   DATA[1200,11] := 2.010372;
   DATA[1200,12] := 0.000256221;
   DATA[1200,13] := 1010.959;
   DATA[1200,14] := 1.0;
   DATA[1200,15] := 1.0;
   DATA[1200,16] := 1.0;
   DATA[1200,17] := 1.0;
   DATA[1200,18] := 1.0;
   DATA[1200,19] := 1.0;
   DATA[1200,20] := 148.808;
   DATA[1200,21] := 154.5501;
   DATA[1200,22] := 1.715439;
   DATA[1200,23] := 841.8226;
   DATA[1200,24] := 2.0;
   DATA[1200,25] := 2.0;
   DATA[1200,26] := 7.87798;
   DATA[1200,27] := 143.5786;
   DATA[1200,28] := 263.0095;
   DATA[1200,29] := 12.07383;
   DATA[1200,30] := 1.725968;
   DATA[1200,31] := 1.253619;
   DATA[1200,32] := 0.7352687;
   DATA[1200,33] := 0.3070813;
   DATA[1200,34] := 2.0;
   DATA[1200,35] := 250.4326;
   DATA[1200,36] := 1.69801;
   DATA[1200,37] := 189.1983;
   DATA[1200,38] := 0.000128152;
   DATA[1200,39] := 1.0;
   DATA[1201,0] := 2.549723;
   DATA[1201,1] := 752.7894;
   DATA[1201,2] := 2.0;
   DATA[1201,3] := 1.0;
   DATA[1201,4] := 262.5288;
   DATA[1201,5] := 8.464369;
   DATA[1201,6] := 317.0982;
   DATA[1201,8] := 1.0;
   DATA[1201,9] := 1.0;
   DATA[1201,10] := 1.0;
   DATA[1201,11] := 2.010372;
   DATA[1201,12] := 0.000256221;
   DATA[1201,13] := 1010.718;
   DATA[1201,14] := 1.0;
   DATA[1201,15] := 1.0;
   DATA[1201,16] := 1.0;
   DATA[1201,17] := 1.0;
   DATA[1201,18] := 1.0;
   DATA[1201,19] := 1.0;
   DATA[1201,20] := 148.808;
   DATA[1201,21] := 154.5501;
   DATA[1201,22] := 1.715952;
   DATA[1201,23] := 842.0149;
   DATA[1201,24] := 2.0;
   DATA[1201,25] := 2.0;
   DATA[1201,26] := 7.87798;
   DATA[1201,27] := 143.5786;
   DATA[1201,28] := 263.0095;
   DATA[1201,29] := 12.07383;
   DATA[1201,30] := 1.725968;
   DATA[1201,31] := 1.261176;
   DATA[1201,32] := 0.7352687;
   DATA[1201,33] := 0.306761;
   DATA[1201,34] := 2.0;
   DATA[1201,35] := 250.4326;
   DATA[1201,36] := 1.69801;
   DATA[1201,37] := 189.1983;
   DATA[1201,38] := 0.000128152;
   DATA[1201,39] := 1.0;
   DATA[1202,0] := 2.551965;
   DATA[1202,1] := 753.2212;
   DATA[1202,2] := 2.0;
   DATA[1202,3] := 1.0;
   DATA[1202,4] := 262.5288;
   DATA[1202,5] := 8.464369;
   DATA[1202,6] := 317.1494;
   DATA[1202,8] := 1.0;
   DATA[1202,9] := 1.0;
   DATA[1202,10] := 1.0;
   DATA[1202,11] := 2.010372;
   DATA[1202,12] := 0.000256221;
   DATA[1202,13] := 1010.839;
   DATA[1202,14] := 1.0;
   DATA[1202,15] := 1.0;
   DATA[1202,16] := 1.0;
   DATA[1202,17] := 1.0;
   DATA[1202,18] := 1.0;
   DATA[1202,19] := 1.0;
   DATA[1202,20] := 148.808;
   DATA[1202,21] := 154.2938;
   DATA[1202,22] := 1.716721;
   DATA[1202,23] := 842.1302;
   DATA[1202,24] := 2.0;
   DATA[1202,25] := 2.0;
   DATA[1202,26] := 7.87798;
   DATA[1202,27] := 143.5786;
   DATA[1202,28] := 263.0095;
   DATA[1202,29] := 12.07383;
   DATA[1202,30] := 1.725968;
   DATA[1202,31] := 1.276803;
   DATA[1202,32] := 0.7352687;
   DATA[1202,33] := 0.3082983;
   DATA[1202,34] := 2.0;
   DATA[1202,35] := 250.4326;
   DATA[1202,36] := 1.69801;
   DATA[1202,37] := 189.2464;
   DATA[1202,38] := 0.000128152;
   DATA[1202,39] := 1.0;
   DATA[1203,0] := 2.551965;
   DATA[1203,1] := 754.0062;
   DATA[1203,2] := 2.0;
   DATA[1203,3] := 1.0;
   DATA[1203,4] := 262.5288;
   DATA[1203,5] := 8.464369;
   DATA[1203,6] := 317.1494;
   DATA[1203,8] := 1.0;
   DATA[1203,9] := 1.0;
   DATA[1203,10] := 1.0;
   DATA[1203,11] := 2.010372;
   DATA[1203,12] := 0.000256221;
   DATA[1203,13] := 1011.079;
   DATA[1203,14] := 1.0;
   DATA[1203,15] := 1.0;
   DATA[1203,16] := 1.0;
   DATA[1203,17] := 1.0;
   DATA[1203,18] := 1.0;
   DATA[1203,19] := 1.0;
   DATA[1203,20] := 148.808;
   DATA[1203,21] := 154.2425;
   DATA[1203,22] := 1.716721;
   DATA[1203,23] := 841.5919;
   DATA[1203,24] := 2.0;
   DATA[1203,25] := 2.0;
   DATA[1203,26] := 7.87798;
   DATA[1203,27] := 143.5786;
   DATA[1203,28] := 263.0095;
   DATA[1203,29] := 12.07383;
   DATA[1203,30] := 1.725968;
   DATA[1203,31] := 1.287562;
   DATA[1203,32] := 0.7352687;
   DATA[1203,33] := 0.3083624;
   DATA[1203,34] := 2.0;
   DATA[1203,35] := 250.4326;
   DATA[1203,36] := 1.69801;
   DATA[1203,37] := 189.2944;
   DATA[1203,38] := 0.000128152;
   DATA[1203,39] := 1.0;
   DATA[1204,0] := 2.554527;
   DATA[1204,1] := 754.1633;
   DATA[1204,2] := 2.0;
   DATA[1204,3] := 1.0;
   DATA[1204,4] := 262.5288;
   DATA[1204,5] := 8.464369;
   DATA[1204,6] := 317.1494;
   DATA[1204,8] := 1.0;
   DATA[1204,9] := 1.0;
   DATA[1204,10] := 1.0;
   DATA[1204,11] := 2.010372;
   DATA[1204,12] := 0.000256221;
   DATA[1204,13] := 1011.119;
   DATA[1204,14] := 1.0;
   DATA[1204,15] := 1.0;
   DATA[1204,16] := 1.0;
   DATA[1204,17] := 1.0;
   DATA[1204,18] := 1.0;
   DATA[1204,19] := 1.0;
   DATA[1204,20] := 148.808;
   DATA[1204,21] := 154.2425;
   DATA[1204,22] := 1.716721;
   DATA[1204,23] := 841.2843;
   DATA[1204,24] := 2.0;
   DATA[1204,25] := 2.0;
   DATA[1204,26] := 7.87798;
   DATA[1204,27] := 143.5786;
   DATA[1204,28] := 263.0095;
   DATA[1204,29] := 12.07383;
   DATA[1204,30] := 1.725968;
   DATA[1204,31] := 1.298578;
   DATA[1204,32] := 0.7352687;
   DATA[1204,33] := 0.3083624;
   DATA[1204,34] := 2.0;
   DATA[1204,35] := 250.4166;
   DATA[1204,36] := 1.69801;
   DATA[1204,37] := 189.2944;
   DATA[1204,38] := 0.000128152;
   DATA[1204,39] := 1.0;
   DATA[1205,0] := 2.554527;
   DATA[1205,1] := 754.2025;
   DATA[1205,2] := 2.0;
   DATA[1205,3] := 1.0;
   DATA[1205,4] := 262.5288;
   DATA[1205,5] := 8.464369;
   DATA[1205,6] := 317.1494;
   DATA[1205,8] := 1.0;
   DATA[1205,9] := 1.0;
   DATA[1205,10] := 1.0;
   DATA[1205,11] := 2.010372;
   DATA[1205,12] := 0.000256221;
   DATA[1205,13] := 1011.079;
   DATA[1205,14] := 1.0;
   DATA[1205,15] := 1.0;
   DATA[1205,16] := 1.0;
   DATA[1205,17] := 1.0;
   DATA[1205,18] := 1.0;
   DATA[1205,19] := 1.0;
   DATA[1205,20] := 148.808;
   DATA[1205,21] := 154.2425;
   DATA[1205,22] := 1.717233;
   DATA[1205,23] := 840.8998;
   DATA[1205,24] := 2.0;
   DATA[1205,25] := 2.0;
   DATA[1205,26] := 7.87798;
   DATA[1205,27] := 143.5786;
   DATA[1205,28] := 263.0095;
   DATA[1205,29] := 12.26609;
   DATA[1205,30] := 1.725968;
   DATA[1205,31] := 1.301396;
   DATA[1205,32] := 0.7352687;
   DATA[1205,33] := 0.3083624;
   DATA[1205,34] := 2.0;
   DATA[1205,35] := 250.2724;
   DATA[1205,36] := 1.69801;
   DATA[1205,37] := 189.1342;
   DATA[1205,38] := 0.000128152;
   DATA[1205,39] := 1.0;
   DATA[1206,0] := 2.554527;
   DATA[1206,1] := 754.7128;
   DATA[1206,2] := 2.0;
   DATA[1206,3] := 1.0;
   DATA[1206,4] := 262.5288;
   DATA[1206,5] := 8.464369;
   DATA[1206,6] := 317.1494;
   DATA[1206,8] := 1.0;
   DATA[1206,9] := 1.0;
   DATA[1206,10] := 1.0;
   DATA[1206,11] := 2.010372;
   DATA[1206,12] := 0.000256221;
   DATA[1206,13] := 1010.919;
   DATA[1206,14] := 1.0;
   DATA[1206,15] := 1.0;
   DATA[1206,16] := 1.0;
   DATA[1206,17] := 1.0;
   DATA[1206,18] := 1.0;
   DATA[1206,19] := 1.0;
   DATA[1206,20] := 148.808;
   DATA[1206,21] := 154.2425;
   DATA[1206,22] := 1.717874;
   DATA[1206,23] := 840.7844;
   DATA[1206,24] := 2.0;
   DATA[1206,25] := 2.0;
   DATA[1206,26] := 7.87798;
   DATA[1206,27] := 143.5786;
   DATA[1206,28] := 263.0095;
   DATA[1206,29] := 12.26609;
   DATA[1206,30] := 1.72443;
   DATA[1206,31] := 1.291789;
   DATA[1206,32] := 0.7352687;
   DATA[1206,33] := 0.3083624;
   DATA[1206,34] := 2.0;
   DATA[1206,35] := 250.2724;
   DATA[1206,36] := 1.69801;
   DATA[1206,37] := 189.0381;
   DATA[1206,38] := 0.000128152;
   DATA[1206,39] := 1.0;
   DATA[1207,0] := 2.554527;
   DATA[1207,1] := 755.2623;
   DATA[1207,2] := 2.0;
   DATA[1207,3] := 1.0;
   DATA[1207,4] := 262.5288;
   DATA[1207,5] := 8.464369;
   DATA[1207,6] := 317.1494;
   DATA[1207,8] := 1.0;
   DATA[1207,9] := 1.0;
   DATA[1207,10] := 1.0;
   DATA[1207,11] := 2.010372;
   DATA[1207,12] := 0.000256221;
   DATA[1207,13] := 1011.159;
   DATA[1207,14] := 1.0;
   DATA[1207,15] := 1.0;
   DATA[1207,16] := 1.0;
   DATA[1207,17] := 1.0;
   DATA[1207,18] := 1.0;
   DATA[1207,19] := 1.0;
   DATA[1207,20] := 148.808;
   DATA[1207,21] := 154.2425;
   DATA[1207,22] := 1.717874;
   DATA[1207,23] := 840.2845;
   DATA[1207,24] := 2.0;
   DATA[1207,25] := 2.0;
   DATA[1207,26] := 7.87798;
   DATA[1207,27] := 143.4248;
   DATA[1207,28] := 263.0095;
   DATA[1207,29] := 12.26609;
   DATA[1207,30] := 1.722892;
   DATA[1207,31] := 1.284232;
   DATA[1207,32] := 0.7352687;
   DATA[1207,33] := 0.3083624;
   DATA[1207,34] := 2.0;
   DATA[1207,35] := 250.1442;
   DATA[1207,36] := 1.69801;
   DATA[1207,37] := 189.0381;
   DATA[1207,38] := 0.000128152;
   DATA[1207,39] := 1.0;
   DATA[1208,0] := 2.55805;
   DATA[1208,1] := 755.6941;
   DATA[1208,2] := 2.0;
   DATA[1208,3] := 1.0;
   DATA[1208,4] := 262.5288;
   DATA[1208,5] := 8.464369;
   DATA[1208,6] := 317.1494;
   DATA[1208,8] := 1.0;
   DATA[1208,9] := 1.0;
   DATA[1208,10] := 1.0;
   DATA[1208,11] := 2.010372;
   DATA[1208,12] := 0.000256221;
   DATA[1208,13] := 1010.718;
   DATA[1208,14] := 1.0;
   DATA[1208,15] := 1.0;
   DATA[1208,16] := 1.0;
   DATA[1208,17] := 1.0;
   DATA[1208,18] := 1.0;
   DATA[1208,19] := 1.0;
   DATA[1208,20] := 148.808;
   DATA[1208,21] := 154.2425;
   DATA[1208,22] := 1.717874;
   DATA[1208,23] := 840.2076;
   DATA[1208,24] := 2.0;
   DATA[1208,25] := 2.0;
   DATA[1208,26] := 7.87798;
   DATA[1208,27] := 143.4248;
   DATA[1208,28] := 263.0095;
   DATA[1208,29] := 12.03538;
   DATA[1208,30] := 1.722892;
   DATA[1208,31] := 1.272576;
   DATA[1208,32] := 0.7352687;
   DATA[1208,33] := 0.3083624;
   DATA[1208,34] := 2.0;
   DATA[1208,35] := 250.1442;
   DATA[1208,36] := 1.69801;
   DATA[1208,37] := 189.0381;
   DATA[1208,38] := 0.000128152;
   DATA[1208,39] := 1.0;
   DATA[1209,0] := 2.559651;
   DATA[1209,1] := 756.4791;
   DATA[1209,2] := 2.0;
   DATA[1209,3] := 1.0;
   DATA[1209,4] := 262.5288;
   DATA[1209,5] := 8.464369;
   DATA[1209,6] := 317.1494;
   DATA[1209,8] := 1.0;
   DATA[1209,9] := 1.0;
   DATA[1209,10] := 1.0;
   DATA[1209,11] := 2.010372;
   DATA[1209,12] := 0.000256221;
   DATA[1209,13] := 1010.919;
   DATA[1209,14] := 1.0;
   DATA[1209,15] := 1.0;
   DATA[1209,16] := 1.0;
   DATA[1209,17] := 1.0;
   DATA[1209,18] := 1.0;
   DATA[1209,19] := 1.0;
   DATA[1209,20] := 148.808;
   DATA[1209,21] := 154.1912;
   DATA[1209,22] := 1.715439;
   DATA[1209,23] := 839.9;
   DATA[1209,24] := 2.0;
   DATA[1209,25] := 2.0;
   DATA[1209,26] := 7.87798;
   DATA[1209,27] := 143.4248;
   DATA[1209,28] := 263.0095;
   DATA[1209,29] := 12.03538;
   DATA[1209,30] := 1.722892;
   DATA[1209,31] := 1.263738;
   DATA[1209,32] := 0.7352687;
   DATA[1209,33] := 0.3083624;
   DATA[1209,34] := 2.0;
   DATA[1209,35] := 250.1442;
   DATA[1209,36] := 1.69801;
   DATA[1209,37] := 189.0381;
   DATA[1209,38] := 0.000128152;
   DATA[1209,39] := 1.0;
   DATA[1210,0] := 2.550043;
   DATA[1210,1] := 756.9502;
   DATA[1210,2] := 2.0;
   DATA[1210,3] := 1.0;
   DATA[1210,4] := 262.5288;
   DATA[1210,5] := 8.464369;
   DATA[1210,6] := 317.1494;
   DATA[1210,8] := 1.0;
   DATA[1210,9] := 1.0;
   DATA[1210,10] := 1.0;
   DATA[1210,11] := 2.010372;
   DATA[1210,12] := 0.000256221;
   DATA[1210,13] := 1010.879;
   DATA[1210,14] := 1.0;
   DATA[1210,15] := 1.0;
   DATA[1210,16] := 1.0;
   DATA[1210,17] := 1.0;
   DATA[1210,18] := 1.0;
   DATA[1210,19] := 1.0;
   DATA[1210,20] := 148.808;
   DATA[1210,21] := 154.0374;
   DATA[1210,22] := 1.713261;
   DATA[1210,23] := 839.2848;
   DATA[1210,24] := 2.0;
   DATA[1210,25] := 2.0;
   DATA[1210,26] := 7.87798;
   DATA[1210,27] := 143.4248;
   DATA[1210,28] := 263.0095;
   DATA[1210,29] := 12.03538;
   DATA[1210,30] := 1.722892;
   DATA[1210,31] := 1.279237;
   DATA[1210,32] := 0.7352687;
   DATA[1210,33] := 0.3083624;
   DATA[1210,34] := 2.0;
   DATA[1210,35] := 250.1442;
   DATA[1210,36] := 1.69801;
   DATA[1210,37] := 189.0381;
   DATA[1210,38] := 0.000128152;
   DATA[1210,39] := 1.0;
   DATA[1211,0] := 2.550043;
   DATA[1211,1] := 757.853;
   DATA[1211,2] := 2.0;
   DATA[1211,3] := 1.0;
   DATA[1211,4] := 262.5288;
   DATA[1211,5] := 8.464369;
   DATA[1211,6] := 317.1494;
   DATA[1211,8] := 1.0;
   DATA[1211,9] := 1.0;
   DATA[1211,10] := 1.0;
   DATA[1211,11] := 2.010372;
   DATA[1211,12] := 0.000256221;
   DATA[1211,13] := 1010.879;
   DATA[1211,14] := 1.0;
   DATA[1211,15] := 1.0;
   DATA[1211,16] := 1.0;
   DATA[1211,17] := 1.0;
   DATA[1211,18] := 1.0;
   DATA[1211,19] := 1.0;
   DATA[1211,20] := 148.808;
   DATA[1211,21] := 153.8836;
   DATA[1211,22] := 1.711723;
   DATA[1211,23] := 839.3232;
   DATA[1211,24] := 2.0;
   DATA[1211,25] := 2.0;
   DATA[1211,26] := 7.87798;
   DATA[1211,27] := 143.4248;
   DATA[1211,28] := 263.0095;
   DATA[1211,29] := 12.03538;
   DATA[1211,30] := 1.722379;
   DATA[1211,31] := 1.289484;
   DATA[1211,32] := 0.7352687;
   DATA[1211,33] := 0.3083624;
   DATA[1211,34] := 2.0;
   DATA[1211,35] := 250.1442;
   DATA[1211,36] := 1.69801;
   DATA[1211,37] := 189.0381;
   DATA[1211,38] := 0.000128152;
   DATA[1211,39] := 1.0;
   DATA[1212,0] := 2.552285;
   DATA[1212,1] := 758.0885;
   DATA[1212,2] := 2.0;
   DATA[1212,3] := 1.0;
   DATA[1212,4] := 262.5288;
   DATA[1212,5] := 8.464369;
   DATA[1212,6] := 317.1494;
   DATA[1212,8] := 1.0;
   DATA[1212,9] := 1.0;
   DATA[1212,10] := 1.0;
   DATA[1212,11] := 2.010372;
   DATA[1212,12] := 0.000256221;
   DATA[1212,13] := 1010.718;
   DATA[1212,14] := 1.0;
   DATA[1212,15] := 1.0;
   DATA[1212,16] := 1.0;
   DATA[1212,17] := 1.0;
   DATA[1212,18] := 1.0;
   DATA[1212,19] := 1.0;
   DATA[1212,20] := 148.808;
   DATA[1212,21] := 153.8836;
   DATA[1212,22] := 1.711082;
   DATA[1212,23] := 838.8618;
   DATA[1212,24] := 2.0;
   DATA[1212,25] := 2.0;
   DATA[1212,26] := 7.87798;
   DATA[1212,27] := 143.4248;
   DATA[1212,28] := 263.0095;
   DATA[1212,29] := 12.03538;
   DATA[1212,30] := 1.722379;
   DATA[1212,31] := 1.299731;
   DATA[1212,32] := 0.7352687;
   DATA[1212,33] := 0.3083624;
   DATA[1212,34] := 2.0;
   DATA[1212,35] := 250.3525;
   DATA[1212,36] := 1.69801;
   DATA[1212,37] := 189.0381;
   DATA[1212,38] := 0.000128152;
   DATA[1212,39] := 1.0;
   DATA[1213,0] := 2.554847;
   DATA[1213,1] := 758.7166;
   DATA[1213,2] := 2.0;
   DATA[1213,3] := 1.0;
   DATA[1213,4] := 262.5288;
   DATA[1213,5] := 8.464369;
   DATA[1213,6] := 317.1494;
   DATA[1213,8] := 1.0;
   DATA[1213,9] := 1.0;
   DATA[1213,10] := 1.0;
   DATA[1213,11] := 2.010372;
   DATA[1213,12] := 0.000256221;
   DATA[1213,13] := 1010.478;
   DATA[1213,14] := 1.0;
   DATA[1213,15] := 1.0;
   DATA[1213,16] := 1.0;
   DATA[1213,17] := 1.0;
   DATA[1213,18] := 1.0;
   DATA[1213,19] := 1.0;
   DATA[1213,20] := 148.808;
   DATA[1213,21] := 153.8836;
   DATA[1213,22] := 1.711082;
   DATA[1213,23] := 838.5542;
   DATA[1213,24] := 2.0;
   DATA[1213,25] := 2.0;
   DATA[1213,26] := 7.87798;
   DATA[1213,27] := 143.4248;
   DATA[1213,28] := 263.0095;
   DATA[1213,29] := 12.03538;
   DATA[1213,30] := 1.722379;
   DATA[1213,31] := 1.30114;
   DATA[1213,32] := 0.7352687;
   DATA[1213,33] := 0.3083624;
   DATA[1213,34] := 2.0;
   DATA[1213,35] := 250.3525;
   DATA[1213,36] := 1.69801;
   DATA[1213,37] := 189.0541;
   DATA[1213,38] := 0.000128152;
   DATA[1213,39] := 1.0;
   DATA[1214,0] := 2.556129;
   DATA[1214,1] := 759.4231;
   DATA[1214,2] := 2.0;
   DATA[1214,3] := 1.0;
   DATA[1214,4] := 262.5288;
   DATA[1214,5] := 8.464369;
   DATA[1214,6] := 317.1494;
   DATA[1214,8] := 1.0;
   DATA[1214,9] := 1.0;
   DATA[1214,10] := 1.0;
   DATA[1214,11] := 2.010372;
   DATA[1214,12] := 0.000256221;
   DATA[1214,13] := 1010.718;
   DATA[1214,14] := 1.0;
   DATA[1214,15] := 1.0;
   DATA[1214,16] := 1.0;
   DATA[1214,17] := 1.0;
   DATA[1214,18] := 1.0;
   DATA[1214,19] := 1.0;
   DATA[1214,20] := 148.808;
   DATA[1214,21] := 154.0118;
   DATA[1214,22] := 1.712363;
   DATA[1214,23] := 838.0543;
   DATA[1214,24] := 2.0;
   DATA[1214,25] := 2.0;
   DATA[1214,26] := 7.87798;
   DATA[1214,27] := 143.3222;
   DATA[1214,28] := 263.0095;
   DATA[1214,29] := 12.03538;
   DATA[1214,30] := 1.725583;
   DATA[1214,31] := 1.291789;
   DATA[1214,32] := 0.7352687;
   DATA[1214,33] := 0.3074656;
   DATA[1214,34] := 2.0;
   DATA[1214,35] := 250.3525;
   DATA[1214,36] := 1.69801;
   DATA[1214,37] := 189.2143;
   DATA[1214,38] := 0.000128152;
   DATA[1214,39] := 1.0;
   DATA[1215,0] := 2.556129;
   DATA[1215,1] := 760.4044;
   DATA[1215,2] := 2.0;
   DATA[1215,3] := 1.0;
   DATA[1215,4] := 262.5288;
   DATA[1215,5] := 8.464369;
   DATA[1215,6] := 317.1494;
   DATA[1215,8] := 1.0;
   DATA[1215,9] := 1.0;
   DATA[1215,10] := 1.0;
   DATA[1215,11] := 2.010372;
   DATA[1215,12] := 0.000256221;
   DATA[1215,13] := 1010.558;
   DATA[1215,14] := 1.0;
   DATA[1215,15] := 1.0;
   DATA[1215,16] := 1.0;
   DATA[1215,17] := 1.0;
   DATA[1215,18] := 1.0;
   DATA[1215,19] := 1.0;
   DATA[1215,20] := 148.808;
   DATA[1215,21] := 154.0118;
   DATA[1215,22] := 1.715567;
   DATA[1215,23] := 837.7852;
   DATA[1215,24] := 2.0;
   DATA[1215,25] := 2.0;
   DATA[1215,26] := 7.87798;
   DATA[1215,27] := 143.2966;
   DATA[1215,28] := 263.0095;
   DATA[1215,29] := 12.03538;
   DATA[1215,30] := 1.72725;
   DATA[1215,31] := 1.282183;
   DATA[1215,32] := 0.7352687;
   DATA[1215,33] := 0.3068891;
   DATA[1215,34] := 2.0;
   DATA[1215,35] := 250.4967;
   DATA[1215,36] := 1.69801;
   DATA[1215,37] := 189.2143;
   DATA[1215,38] := 0.000128152;
   DATA[1215,39] := 1.0;
   DATA[1216,0] := 2.553566;
   DATA[1216,1] := 760.9932;
   DATA[1216,2] := 2.0;
   DATA[1216,3] := 1.0;
   DATA[1216,4] := 262.5288;
   DATA[1216,5] := 8.464369;
   DATA[1216,6] := 317.1494;
   DATA[1216,8] := 1.0;
   DATA[1216,9] := 1.0;
   DATA[1216,10] := 1.0;
   DATA[1216,11] := 2.010372;
   DATA[1216,12] := 0.000256221;
   DATA[1216,13] := 1010.959;
   DATA[1216,14] := 1.0;
   DATA[1216,15] := 1.0;
   DATA[1216,16] := 1.0;
   DATA[1216,17] := 1.0;
   DATA[1216,18] := 1.0;
   DATA[1216,19] := 1.0;
   DATA[1216,20] := 148.808;
   DATA[1216,21] := 154.0118;
   DATA[1216,22] := 1.716721;
   DATA[1216,23] := 837.2853;
   DATA[1216,24] := 2.0;
   DATA[1216,25] := 2.0;
   DATA[1216,26] := 7.87798;
   DATA[1216,27] := 143.2966;
   DATA[1216,28] := 263.0095;
   DATA[1216,29] := 12.03538;
   DATA[1216,30] := 1.727378;
   DATA[1216,31] := 1.273857;
   DATA[1216,32] := 0.7352687;
   DATA[1216,33] := 0.3068891;
   DATA[1216,34] := 2.0;
   DATA[1216,35] := 250.4967;
   DATA[1216,36] := 1.69801;
   DATA[1216,37] := 189.2624;
   DATA[1216,38] := 0.000128152;
   DATA[1216,39] := 1.0;
   DATA[1217,0] := 2.550684;
   DATA[1217,1] := 761.3465;
   DATA[1217,2] := 2.0;
   DATA[1217,3] := 1.0;
   DATA[1217,4] := 262.5288;
   DATA[1217,5] := 8.464369;
   DATA[1217,6] := 317.2263;
   DATA[1217,8] := 1.0;
   DATA[1217,9] := 1.0;
   DATA[1217,10] := 1.0;
   DATA[1217,11] := 2.010372;
   DATA[1217,12] := 0.000256221;
   DATA[1217,13] := 1010.758;
   DATA[1217,14] := 1.0;
   DATA[1217,15] := 1.0;
   DATA[1217,16] := 1.0;
   DATA[1217,17] := 1.0;
   DATA[1217,18] := 1.0;
   DATA[1217,19] := 1.0;
   DATA[1217,20] := 148.808;
   DATA[1217,21] := 154.0118;
   DATA[1217,22] := 1.716849;
   DATA[1217,23] := 837.516;
   DATA[1217,24] := 2.0;
   DATA[1217,25] := 2.0;
   DATA[1217,26] := 7.87798;
   DATA[1217,27] := 143.2966;
   DATA[1217,28] := 263.0095;
   DATA[1217,29] := 12.03538;
   DATA[1217,30] := 1.727378;
   DATA[1217,31] := 1.287947;
   DATA[1217,32] := 0.7352687;
   DATA[1217,33] := 0.3068891;
   DATA[1217,34] := 2.0;
   DATA[1217,35] := 250.5127;
   DATA[1217,36] := 1.69801;
   DATA[1217,37] := 189.2624;
   DATA[1217,38] := 0.000128152;
   DATA[1217,39] := 1.0;
   DATA[1218,0] := 2.550684;
   DATA[1218,1] := 762.524;
   DATA[1218,2] := 2.0;
   DATA[1218,3] := 1.0;
   DATA[1218,4] := 262.5288;
   DATA[1218,5] := 8.464369;
   DATA[1218,6] := 317.2263;
   DATA[1218,8] := 1.0;
   DATA[1218,9] := 1.0;
   DATA[1218,10] := 1.0;
   DATA[1218,11] := 2.010372;
   DATA[1218,12] := 0.000256221;
   DATA[1218,13] := 1010.718;
   DATA[1218,14] := 1.0;
   DATA[1218,15] := 1.0;
   DATA[1218,16] := 1.0;
   DATA[1218,17] := 1.0;
   DATA[1218,18] := 1.0;
   DATA[1218,19] := 1.0;
   DATA[1218,20] := 148.808;
   DATA[1218,21] := 154.0118;
   DATA[1218,22] := 1.716849;
   DATA[1218,23] := 837.17;
   DATA[1218,24] := 2.0;
   DATA[1218,25] := 2.0;
   DATA[1218,26] := 7.87798;
   DATA[1218,27] := 143.2966;
   DATA[1218,28] := 263.0095;
   DATA[1218,29] := 12.03538;
   DATA[1218,30] := 1.727378;
   DATA[1218,31] := 1.3005;
   DATA[1218,32] := 0.7352687;
   DATA[1218,33] := 0.3066329;
   DATA[1218,34] := 2.0;
   DATA[1218,35] := 250.5127;
   DATA[1218,36] := 1.69801;
   DATA[1218,37] := 189.3745;
   DATA[1218,38] := 0.000128152;
   DATA[1218,39] := 1.0;
   DATA[1219,0] := 2.551324;
   DATA[1219,1] := 762.8381;
   DATA[1219,2] := 2.0;
   DATA[1219,3] := 1.0;
   DATA[1219,4] := 262.5288;
   DATA[1219,5] := 8.464369;
   DATA[1219,6] := 317.2263;
   DATA[1219,8] := 1.0;
   DATA[1219,9] := 1.0;
   DATA[1219,10] := 1.0;
   DATA[1219,11] := 2.010372;
   DATA[1219,12] := 0.000256221;
   DATA[1219,13] := 1010.879;
   DATA[1219,14] := 1.0;
   DATA[1219,15] := 1.0;
   DATA[1219,16] := 1.0;
   DATA[1219,17] := 1.0;
   DATA[1219,18] := 1.0;
   DATA[1219,19] := 1.0;
   DATA[1219,20] := 148.808;
   DATA[1219,21] := 154.0118;
   DATA[1219,22] := 1.717233;
   DATA[1219,23] := 836.6317;
   DATA[1219,24] := 2.0;
   DATA[1219,25] := 2.0;
   DATA[1219,26] := 7.87798;
   DATA[1219,27] := 143.2966;
   DATA[1219,28] := 263.0095;
   DATA[1219,29] := 12.03538;
   DATA[1219,30] := 1.728531;
   DATA[1219,31] := 1.302037;
   DATA[1219,32] := 0.7352687;
   DATA[1219,33] := 0.3066329;
   DATA[1219,34] := 2.0;
   DATA[1219,35] := 250.5127;
   DATA[1219,36] := 1.69801;
   DATA[1219,37] := 189.3745;
   DATA[1219,38] := 0.000128152;
   DATA[1219,39] := 1.0;
   DATA[1220,0] := 2.551324;
   DATA[1220,1] := 763.5839;
   DATA[1220,2] := 2.0;
   DATA[1220,3] := 1.0;
   DATA[1220,4] := 262.5288;
   DATA[1220,5] := 8.464369;
   DATA[1220,6] := 317.2263;
   DATA[1220,8] := 1.0;
   DATA[1220,9] := 1.0;
   DATA[1220,10] := 1.0;
   DATA[1220,11] := 2.010372;
   DATA[1220,12] := 0.000256221;
   DATA[1220,13] := 1010.839;
   DATA[1220,14] := 1.0;
   DATA[1220,15] := 1.0;
   DATA[1220,16] := 1.0;
   DATA[1220,17] := 1.0;
   DATA[1220,18] := 1.0;
   DATA[1220,19] := 1.0;
   DATA[1220,20] := 148.808;
   DATA[1220,21] := 154.0118;
   DATA[1220,22] := 1.717489;
   DATA[1220,23] := 836.2471;
   DATA[1220,24] := 2.0;
   DATA[1220,25] := 2.0;
   DATA[1220,26] := 7.87798;
   DATA[1220,27] := 143.2966;
   DATA[1220,28] := 263.0095;
   DATA[1220,29] := 12.26609;
   DATA[1220,30] := 1.728531;
   DATA[1220,31] := 1.302037;
   DATA[1220,32] := 0.7352687;
   DATA[1220,33] := 0.3066329;
   DATA[1220,34] := 2.0;
   DATA[1220,35] := 250.5127;
   DATA[1220,36] := 1.69801;
   DATA[1220,37] := 189.3745;
   DATA[1220,38] := 0.000128152;
   DATA[1220,39] := 1.0;
   DATA[1221,0] := 2.543958;
   DATA[1221,1] := 764.212;
   DATA[1221,2] := 2.0;
   DATA[1221,3] := 1.0;
   DATA[1221,4] := 262.5288;
   DATA[1221,5] := 8.464369;
   DATA[1221,6] := 317.2263;
   DATA[1221,8] := 1.0;
   DATA[1221,9] := 1.0;
   DATA[1221,10] := 1.0;
   DATA[1221,11] := 2.010372;
   DATA[1221,12] := 0.000256221;
   DATA[1221,13] := 1010.839;
   DATA[1221,14] := 1.0;
   DATA[1221,15] := 1.0;
   DATA[1221,16] := 1.0;
   DATA[1221,17] := 1.0;
   DATA[1221,18] := 1.0;
   DATA[1221,19] := 1.0;
   DATA[1221,20] := 148.808;
   DATA[1221,21] := 154.2425;
   DATA[1221,22] := 1.717489;
   DATA[1221,23] := 835.978;
   DATA[1221,24] := 2.0;
   DATA[1221,25] := 2.0;
   DATA[1221,26] := 7.87798;
   DATA[1221,27] := 143.2966;
   DATA[1221,28] := 263.0095;
   DATA[1221,29] := 12.26609;
   DATA[1221,30] := 1.728531;
   DATA[1221,31] := 1.30178;
   DATA[1221,32] := 0.7352687;
   DATA[1221,33] := 0.3066329;
   DATA[1221,34] := 2.0;
   DATA[1221,35] := 250.5127;
   DATA[1221,36] := 1.69801;
   DATA[1221,37] := 189.3745;
   DATA[1221,38] := 0.000128152;
   DATA[1221,39] := 1.0;
   DATA[1222,0] := 2.543638;
   DATA[1222,1] := 765.154;
   DATA[1222,2] := 2.0;
   DATA[1222,3] := 1.0;
   DATA[1222,4] := 262.5288;
   DATA[1222,5] := 8.464369;
   DATA[1222,6] := 317.2263;
   DATA[1222,8] := 1.0;
   DATA[1222,9] := 1.0;
   DATA[1222,10] := 1.0;
   DATA[1222,11] := 2.010372;
   DATA[1222,12] := 0.000256221;
   DATA[1222,13] := 1010.678;
   DATA[1222,14] := 1.0;
   DATA[1222,15] := 1.0;
   DATA[1222,16] := 1.0;
   DATA[1222,17] := 1.0;
   DATA[1222,18] := 1.0;
   DATA[1222,19] := 1.0;
   DATA[1222,20] := 148.808;
   DATA[1222,21] := 154.2425;
   DATA[1222,22] := 1.71467;
   DATA[1222,23] := 835.3627;
   DATA[1222,24] := 2.0;
   DATA[1222,25] := 2.0;
   DATA[1222,26] := 7.87798;
   DATA[1222,27] := 143.2966;
   DATA[1222,28] := 263.0095;
   DATA[1222,29] := 11.95847;
   DATA[1222,30] := 1.728531;
   DATA[1222,31] := 1.291405;
   DATA[1222,32] := 0.7352687;
   DATA[1222,33] := 0.3066329;
   DATA[1222,34] := 2.0;
   DATA[1222,35] := 250.5127;
   DATA[1222,36] := 1.69801;
   DATA[1222,37] := 189.3745;
   DATA[1222,38] := 0.000128152;
   DATA[1222,39] := 1.0;
   DATA[1223,0] := 2.547161;
   DATA[1223,1] := 765.154;
   DATA[1223,2] := 2.0;
   DATA[1223,3] := 1.0;
   DATA[1223,4] := 262.5288;
   DATA[1223,5] := 8.464369;
   DATA[1223,6] := 317.2263;
   DATA[1223,8] := 1.0;
   DATA[1223,9] := 1.0;
   DATA[1223,10] := 1.0;
   DATA[1223,11] := 2.010372;
   DATA[1223,12] := 0.000256221;
   DATA[1223,13] := 1010.678;
   DATA[1223,14] := 1.0;
   DATA[1223,15] := 1.0;
   DATA[1223,16] := 1.0;
   DATA[1223,17] := 1.0;
   DATA[1223,18] := 1.0;
   DATA[1223,19] := 1.0;
   DATA[1223,20] := 148.808;
   DATA[1223,21] := 154.2425;
   DATA[1223,22] := 1.71262;
   DATA[1223,23] := 834.8244;
   DATA[1223,24] := 2.0;
   DATA[1223,25] := 2.0;
   DATA[1223,26] := 7.87798;
   DATA[1223,27] := 143.2966;
   DATA[1223,28] := 263.1056;
   DATA[1223,29] := 11.95847;
   DATA[1223,30] := 1.726609;
   DATA[1223,31] := 1.291405;
   DATA[1223,32] := 0.7352687;
   DATA[1223,33] := 0.3066329;
   DATA[1223,34] := 2.0;
   DATA[1223,35] := 250.5127;
   DATA[1223,36] := 1.69801;
   DATA[1223,37] := 189.3745;
   DATA[1223,38] := 0.000128152;
   DATA[1223,39] := 1.0;
   DATA[1224,0] := 2.556449;
   DATA[1224,1] := 765.7036;
   DATA[1224,2] := 2.0;
   DATA[1224,3] := 1.0;
   DATA[1224,4] := 262.5288;
   DATA[1224,5] := 8.464369;
   DATA[1224,6] := 317.2263;
   DATA[1224,8] := 1.0;
   DATA[1224,9] := 1.0;
   DATA[1224,10] := 1.0;
   DATA[1224,11] := 2.010372;
   DATA[1224,12] := 0.000256221;
   DATA[1224,13] := 1011.039;
   DATA[1224,14] := 1.0;
   DATA[1224,15] := 1.0;
   DATA[1224,16] := 1.0;
   DATA[1224,17] := 1.0;
